;ENDFOLD
;FOLD CIRC CAux389 CDes389 CONT Vel=0.1 m/s CPDATC389 Tool[2] Base[10] ;%{PE}
;FOLD Parameters ;%{h}
;Params IlfProvider=kukaroboter.basistech.inlineforms.movement.old; Kuka.IsGlobalPoint=False; Kuka.PointName=CDes389; Kuka.BlendingEnabled=TRUE; Kuka.MoveDataName=CPDATC389; Kuka.VelocityPath=0.1; Kuka.CurrentCDSetIndex=0; Kuka.MovementParameterFieldEnabled=True; IlfCommand=LIN
;ENDFOLD
$BWDSTART = FALSE
LDAT_ACT=LCPDATC389
FDAT_ACT=FC389
$ORI_TYPE = #VAR
$CIRC_TYPE = #PATH
BAS (#CP_PARAMS,0.1)
SET_CD_PARAMS (0)
CIRC XCAux389, XCDes389 C_DIS

;ENDFOLD
;FOLD LIN P390 CONT Vel=1 m/s CPDATP390 Tool[2] Base[10] ;%{PE}
;FOLD Parameters ;%{h}
;Params IlfProvider=kukaroboter.basistech.inlineforms.movement.old; Kuka.IsGlobalPoint=False; Kuka.PointName=P390; Kuka.BlendingEnabled=TRUE; Kuka.MoveDataName=CPDATP390; Kuka.VelocityPath=1; Kuka.CurrentCDSetIndex=0; Kuka.MovementParameterFieldEnabled=True; IlfCommand=LIN
;ENDFOLD
$BWDSTART = FALSE
LDAT_ACT=LCPDATP390
FDAT_ACT=FP390
BAS (#CP_PARAMS,1)
SET_CD_PARAMS (0)
LIN XP390 C_DIS

;ENDFOLD
;FOLD LIN P391 CONT Vel=1 m/s CPDATP391 Tool[2] Base[10] ;%{PE}
;FOLD Parameters ;%{h}
;Params IlfProvider=kukaroboter.basistech.inlineforms.movement.old; Kuka.IsGlobalPoint=False; Kuka.PointName=P391; Kuka.BlendingEnabled=TRUE; Kuka.MoveDataName=CPDATP391; Kuka.VelocityPath=1; Kuka.CurrentCDSetIndex=0; Kuka.MovementParameterFieldEnabled=True; IlfCommand=LIN
;ENDFOLD
$BWDSTART = FALSE
LDAT_ACT=LCPDATP391
FDAT_ACT=FP391
BAS (#CP_PARAMS,1)
SET_CD_PARAMS (0)
LIN XP391 C_DIS

;ENDFOLD
;FOLD CIRC CAux392 CDes392 CONT Vel=0.1 m/s CPDATC392 Tool[2] Base[10] ;%{PE}
;FOLD Parameters ;%{h}
;Params IlfProvider=kukaroboter.basistech.inlineforms.movement.old; Kuka.IsGlobalPoint=False; Kuka.PointName=CDes392; Kuka.BlendingEnabled=TRUE; Kuka.MoveDataName=CPDATC392; Kuka.VelocityPath=0.1; Kuka.CurrentCDSetIndex=0; Kuka.MovementParameterFieldEnabled=True; IlfCommand=LIN
;ENDFOLD
$BWDSTART = FALSE
LDAT_ACT=LCPDATC392
FDAT_ACT=FC392
$ORI_TYPE = #VAR
$CIRC_TYPE = #PATH
BAS (#CP_PARAMS,0.1)
SET_CD_PARAMS (0)
CIRC XCAux392, XCDes392 C_DIS

;ENDFOLD
;FOLD LIN P393 CONT Vel=1 m/s CPDATP393 Tool[2] Base[10] ;%{PE}
;FOLD Parameters ;%{h}
;Params IlfProvider=kukaroboter.basistech.inlineforms.movement.old; Kuka.IsGlobalPoint=False; Kuka.PointName=P393; Kuka.BlendingEnabled=TRUE; Kuka.MoveDataName=CPDATP393; Kuka.VelocityPath=1; Kuka.CurrentCDSetIndex=0; Kuka.MovementParameterFieldEnabled=True; IlfCommand=LIN
;ENDFOLD
$BWDSTART = FALSE
LDAT_ACT=LCPDATP393
FDAT_ACT=FP393
BAS (#CP_PARAMS,1)
SET_CD_PARAMS (0)
LIN XP393 C_DIS

;ENDFOLD
;FOLD LIN P394 CONT Vel=1 m/s CPDATP394 Tool[2] Base[10] ;%{PE}
;FOLD Parameters ;%{h}
;Params IlfProvider=kukaroboter.basistech.inlineforms.movement.old; Kuka.IsGlobalPoint=False; Kuka.PointName=P394; Kuka.BlendingEnabled=TRUE; Kuka.MoveDataName=CPDATP394; Kuka.VelocityPath=1; Kuka.CurrentCDSetIndex=0; Kuka.MovementParameterFieldEnabled=True; IlfCommand=LIN
;ENDFOLD
$BWDSTART = FALSE
LDAT_ACT=LCPDATP394
FDAT_ACT=FP394
BAS (#CP_PARAMS,1)
SET_CD_PARAMS (0)
LIN XP394 C_DIS

;ENDFOLD
;FOLD CIRC CAux395 CDes395 CONT Vel=0.1 m/s CPDATC395 Tool[2] Base[10] ;%{PE}
;FOLD Parameters ;%{h}
;Params IlfProvider=kukaroboter.basistech.inlineforms.movement.old; Kuka.IsGlobalPoint=False; Kuka.PointName=CDes395; Kuka.BlendingEnabled=TRUE; Kuka.MoveDataName=CPDATC395; Kuka.VelocityPath=0.1; Kuka.CurrentCDSetIndex=0; Kuka.MovementParameterFieldEnabled=True; IlfCommand=LIN
;ENDFOLD
$BWDSTART = FALSE
LDAT_ACT=LCPDATC395
FDAT_ACT=FC395
$ORI_TYPE = #VAR
$CIRC_TYPE = #PATH
BAS (#CP_PARAMS,0.1)
SET_CD_PARAMS (0)
CIRC XCAux395, XCDes395 C_DIS

;ENDFOLD
;FOLD LIN P396 CONT Vel=1 m/s CPDATP396 Tool[2] Base[10] ;%{PE}
;FOLD Parameters ;%{h}
;Params IlfProvider=kukaroboter.basistech.inlineforms.movement.old; Kuka.IsGlobalPoint=False; Kuka.PointName=P396; Kuka.BlendingEnabled=TRUE; Kuka.MoveDataName=CPDATP396; Kuka.VelocityPath=1; Kuka.CurrentCDSetIndex=0; Kuka.MovementParameterFieldEnabled=True; IlfCommand=LIN
;ENDFOLD
$BWDSTART = FALSE
LDAT_ACT=LCPDATP396
FDAT_ACT=FP396
BAS (#CP_PARAMS,1)
SET_CD_PARAMS (0)
LIN XP396 C_DIS

;ENDFOLD
;FOLD LIN P397 CONT Vel=0.5 m/s CPDATP397 Tool[2] Base[10] ;%{PE}
;FOLD Parameters ;%{h}
;Params IlfProvider=kukaroboter.basistech.inlineforms.movement.old; Kuka.IsGlobalPoint=False; Kuka.PointName=P397; Kuka.BlendingEnabled=TRUE; Kuka.MoveDataName=CPDATP397; Kuka.VelocityPath=0.5; Kuka.CurrentCDSetIndex=0; Kuka.MovementParameterFieldEnabled=True; IlfCommand=LIN
;ENDFOLD
$BWDSTART = FALSE
LDAT_ACT=LCPDATP397
FDAT_ACT=FP397
BAS (#CP_PARAMS,0.5)
SET_CD_PARAMS (0)
LIN XP397 C_DIS

;ENDFOLD
;FOLD LIN P398 CONT Vel=0.5 m/s CPDATP398 Tool[2] Base[10] ;%{PE}
;FOLD Parameters ;%{h}
;Params IlfProvider=kukaroboter.basistech.inlineforms.movement.old; Kuka.IsGlobalPoint=False; Kuka.PointName=P398; Kuka.BlendingEnabled=TRUE; Kuka.MoveDataName=CPDATP398; Kuka.VelocityPath=0.5; Kuka.CurrentCDSetIndex=0; Kuka.MovementParameterFieldEnabled=True; IlfCommand=LIN
;ENDFOLD
$BWDSTART = FALSE
LDAT_ACT=LCPDATP398
FDAT_ACT=FP398
BAS (#CP_PARAMS,0.5)
SET_CD_PARAMS (0)
LIN XP398 C_DIS

;ENDFOLD
;FOLD LIN P399 CONT Vel=1.0 m/s CPDATP399 Tool[2] Base[10] ;%{PE}
;FOLD Parameters ;%{h}
;Params IlfProvider=kukaroboter.basistech.inlineforms.movement.old; Kuka.IsGlobalPoint=False; Kuka.PointName=P399; Kuka.BlendingEnabled=TRUE; Kuka.MoveDataName=CPDATP399; Kuka.VelocityPath=1.0; Kuka.CurrentCDSetIndex=0; Kuka.MovementParameterFieldEnabled=True; IlfCommand=LIN
;ENDFOLD
$BWDSTART = FALSE
LDAT_ACT=LCPDATP399
FDAT_ACT=FP399
BAS (#CP_PARAMS,1.0)
SET_CD_PARAMS (0)
LIN XP399 C_DIS

;ENDFOLD
;FOLD LIN P400 CONT Vel=1.0 m/s CPDATP400 Tool[2] Base[10] ;%{PE}
;FOLD Parameters ;%{h}
;Params IlfProvider=kukaroboter.basistech.inlineforms.movement.old; Kuka.IsGlobalPoint=False; Kuka.PointName=P400; Kuka.BlendingEnabled=TRUE; Kuka.MoveDataName=CPDATP400; Kuka.VelocityPath=1.0; Kuka.CurrentCDSetIndex=0; Kuka.MovementParameterFieldEnabled=True; IlfCommand=LIN
;ENDFOLD
$BWDSTART = FALSE
LDAT_ACT=LCPDATP400
FDAT_ACT=FP400
BAS (#CP_PARAMS,1.0)
SET_CD_PARAMS (0)
LIN XP400 C_DIS

;ENDFOLD
END
;End of routine {i}

--- repair_test.dat ---
&ACCESS RVP1
&REL 1217
&PARAM WOPTRAJECTORYID = 2
&PARAM WOPTEMPLATENAME = WopCoreTemplatePath
&PARAM DISKPATH = KRC:\R1\Program\Working Paths
DEFDAT  repair_test
;FOLD EXTERNAL DECLARATIONS;%{PE}%MKUKATPBASIS,%CEXT,%VCOMMON,%P
;FOLD BASISTECH EXT;%{PE}%MKUKATPBASIS,%CEXT,%VEXT,%P
EXT  BAS (BAS_COMMAND  :IN,REAL  :IN )
DECL INT SUCCESS
;ENDFOLD (BASISTECH EXT)
;FOLD USER EXT;%{E}%MKUKATPUSER,%CEXT,%VEXT,%P
;Make your modifications here

;ENDFOLD (USER EXT)
;ENDFOLD (EXTERNAL DECLARATIONS)

INT APP_GENNUMBER = 215375
INT APP_ANSWER
INT APP_OFFSET
DECL STATE_T APP_STATE

DECL PDAT PPDATP0={VEL 100,ACC 100,APO_DIST 5,APO_MODE #CDIS,GEAR_JERK 100.0,EXAX_IGN 0}
DECL FDAT FP0={TOOL_NO 2,BASE_NO 10,IPO_FRAME #BASE,POINT2[] " ",TQ_STATE FALSE}
DECL E6AXIS XP0={A1 -1000.000,A2 -90.000,A3 90.000,A4 0.000,A5 -90.000,A6 0.000,E1 0.000,E2 -41.000,E3 33.000,E4 0.000,E5 0.000,E6 0.000}

; Data for Routine_0
DECL LDAT LCPDATP1={VEL 1,ACC 100,APO_DIST 5,APO_FAC 50.0,ORI_TYP #VAR,CIRC_TYP #BASE,JERK_FAC 50.0}
DECL FDAT FP1={TOOL_NO 2,BASE_NO 10,IPO_FRAME #BASE,POINT2[] " ",TQ_STATE FALSE}
DECL E6POS XP1={X -60.500,Y 111.430,Z -37.190,A 0.000,B -17.860,C -36.410}
DECL LDAT LCPDATC2={VEL 0.1,ACC 100,APO_DIST 5,APO_FAC 50.0,ORI_TYP #VAR,CIRC_TYP #BASE,JERK_FAC 50.0}
DECL FDAT FC2={TOOL_NO 2,BASE_NO 10,IPO_FRAME #BASE,POINT2[] " ",TQ_STATE FALSE}
DECL E6POS XCAux2={X -48.520,Y 117.140,Z -37.190,A 0.000,B -14.240,C -37.780}
DECL E6POS XCDes2={X 48.520,Y 117.140,Z -37.190,A 0.000,B 14.240,C -37.780}
DECL LDAT LCPDATP3={VEL 1,ACC 100,APO_DIST 5,APO_FAC 50.0,ORI_TYP #VAR,CIRC_TYP #BASE,JERK_FAC 50.0}
DECL FDAT FP3={TOOL_NO 2,BASE_NO 10,IPO_FRAME #BASE,POINT2[] " ",TQ_STATE FALSE}
DECL E6POS XP3={X 60.500,Y 111.430,Z -37.190,A 0.000,B 17.860,C -36.410}
DECL LDAT LCPDATP4={VEL 1,ACC 100,APO_DIST 5,APO_FAC 50.0,ORI_TYP #VAR,CIRC_TYP #BASE,JERK_FAC 50.0}
DECL FDAT FP4={TOOL_NO 2,BASE_NO 10,IPO_FRAME #BASE,POINT2[] " ",TQ_STATE FALSE}
DECL E6POS XP4={X 62.870,Y 115.800,Z -40.720,A 0.000,B 14.110,C -27.570}
DECL LDAT LCPDATC5={VEL 0.1,ACC 100,APO_DIST 5,APO_FAC 50.0,ORI_TYP #VAR,CIRC_TYP #BASE,JERK_FAC 50.0}
DECL FDAT FC5={TOOL_NO 2,BASE_NO 10,IPO_FRAME #BASE,POINT2[] " ",TQ_STATE FALSE}
DECL E6POS XCAux5={X 50.420,Y 121.740,Z -40.720,A 0.000,B 11.270,C -28.760}
DECL E6POS XCDes5={X -50.420,Y 121.740,Z -40.720,A 0.000,B -11.270,C -28.760}
DECL LDAT LCPDATP6={VEL 1,ACC 100,APO_DIST 5,APO_FAC 50.0,ORI_TYP #VAR,CIRC_TYP #BASE,JERK_FAC 50.0}
DECL FDAT FP6={TOOL_NO 2,BASE_NO 10,IPO_FRAME #BASE,POINT2[] " ",TQ_STATE FALSE}
DECL E6POS XP6={X -62.870,Y 115.800,Z -40.720,A -0.000,B -14.110,C -27.570}
DECL LDAT LCPDATP7={VEL 1,ACC 100,APO_DIST 5,APO_FAC 50.0,ORI_TYP #VAR,CIRC_TYP #BASE,JERK_FAC 50.0}
DECL FDAT FP7={TOOL_NO 2,BASE_NO 10,IPO_FRAME #BASE,POINT2[] " ",TQ_STATE FALSE}
DECL E6POS XP7={X -65.490,Y 120.610,Z -43.400,A 0.000,B -10.040,C -19.030}
DECL LDAT LCPDATC8={VEL 0.1,ACC 100,APO_DIST 5,APO_FAC 50.0,ORI_TYP #VAR,CIRC_TYP #BASE,JERK_FAC 50.0}
DECL FDAT FC8={TOOL_NO 2,BASE_NO 10,IPO_FRAME #BASE,POINT2[] " ",TQ_STATE FALSE}
DECL E6POS XCAux8={X -52.520,Y 126.790,Z -43.400,A 0.000,B -8.040,C -19.930}
DECL E6POS XCDes8={X 52.520,Y 126.790,Z -43.400,A 0.000,B 8.040,C -19.930}
DECL LDAT LCPDATP9={VEL 1,ACC 100,APO_DIST 5,APO_FAC 50.0,ORI_TYP #VAR,CIRC_TYP #BASE,JERK_FAC 50.0}
DECL FDAT FP9={TOOL_NO 2,BASE_NO 10,IPO_FRAME #BASE,POINT2[] " ",TQ_STATE FALSE}
DECL E6POS XP9={X 65.490,Y 120.610,Z -43.400,A 0.000,B 10.040,C -19.030}
DECL LDAT LCPDATP10={VEL 1,ACC 100,APO_DIST 5,APO_FAC 50.0,ORI_TYP #VAR,CIRC_TYP #BASE,JERK_FAC 50.0}
DECL FDAT FP10={TOOL_NO 2,BASE_NO 10,IPO_FRAME #BASE,POINT2[] " ",TQ_STATE FALSE}
DECL E6POS XP10={X 68.270,Y 125.740,Z -45.160,A -0.000,B 5.760,C -10.710}
DECL LDAT LCPDATC11={VEL 0.1,ACC 100,APO_DIST 5,APO_FAC 50.0,ORI_TYP #VAR,CIRC_TYP #BASE,JERK_FAC 50.0}
DECL FDAT FC11={TOOL_NO 2,BASE_NO 10,IPO_FRAME #BASE,POINT2[] " ",TQ_STATE FALSE}
DECL E6POS XCAux11={X 54.750,Y 132.190,Z -45.160,A -0.000,B 4.620,C -11.250}
DECL E6POS XCDes11={X -54.750,Y 132.190,Z -45.160,A 0.000,B -4.620,C -11.250}
DECL LDAT LCPDATP12={VEL 1,ACC 100,APO_DIST 5,APO_FAC 50.0,ORI_TYP #VAR,CIRC_TYP #BASE,JERK_FAC 50.0}
DECL FDAT FP12={TOOL_NO 2,BASE_NO 10,IPO_FRAME #BASE,POINT2[] " ",TQ_STATE FALSE}
DECL E6POS XP12={X -68.270,Y 125.740,Z -45.160,A 0.000,B -5.760,C -10.710}
DECL LDAT LCPDATP13={VEL 1,ACC 100,APO_DIST 5,APO_FAC 50.0,ORI_TYP #VAR,CIRC_TYP #BASE,JERK_FAC 50.0}
DECL FDAT FP13={TOOL_NO 2,BASE_NO 10,IPO_FRAME #BASE,POINT2[] " ",TQ_STATE FALSE}
DECL E6POS XP13={X -71.150,Y 131.050,Z -45.950,A 0.000,B -1.370,C -2.520}
DECL LDAT LCPDATC14={VEL 0.1,ACC 100,APO_DIST 5,APO_FAC 50.0,ORI_TYP #VAR,CIRC_TYP #BASE,JERK_FAC 50.0}
DECL FDAT FC14={TOOL_NO 2,BASE_NO 10,IPO_FRAME #BASE,POINT2[] " ",TQ_STATE FALSE}
DECL E6POS XCAux14={X -57.070,Y 137.770,Z -45.950,A 0.000,B -1.090,C -2.640}
DECL E6POS XCDes14={X 57.070,Y 137.770,Z -45.950,A -0.000,B 1.090,C -2.640}
DECL LDAT LCPDATP15={VEL 1,ACC 100,APO_DIST 5,APO_FAC 50.0,ORI_TYP #VAR,CIRC_TYP #BASE,JERK_FAC 50.0}
DECL FDAT FP15={TOOL_NO 2,BASE_NO 10,IPO_FRAME #BASE,POINT2[] " ",TQ_STATE FALSE}
DECL E6POS XP15={X 71.150,Y 131.050,Z -45.950,A 0.000,B 1.370,C -2.520}
DECL LDAT LCPDATP16={VEL 1,ACC 100,APO_DIST 5,APO_FAC 50.0,ORI_TYP #VAR,CIRC_TYP #BASE,JERK_FAC 50.0}
DECL FDAT FP16={TOOL_NO 2,BASE_NO 10,IPO_FRAME #BASE,POINT2[] " ",TQ_STATE FALSE}
DECL E6POS XP16={X 71.390,Y 131.490,Z -46.000,A 0.000,B 0.000,C -0.000}
DECL LDAT LCPDATC17={VEL 0.1,ACC 100,APO_DIST 5,APO_FAC 50.0,ORI_TYP #VAR,CIRC_TYP #BASE,JERK_FAC 50.0}
DECL FDAT FC17={TOOL_NO 2,BASE_NO 10,IPO_FRAME #BASE,POINT2[] " ",TQ_STATE FALSE}
DECL E6POS XCAux17={X 57.260,Y 138.230,Z -46.000,A 0.000,B 0.000,C -0.000}
DECL E6POS XCDes17={X -57.260,Y 138.230,Z -46.000,A 0.000,B 0.000,C -0.000}
DECL LDAT LCPDATP18={VEL 1,ACC 100,APO_DIST 5,APO_FAC 50.0,ORI_TYP #VAR,CIRC_TYP #BASE,JERK_FAC 50.0}
DECL FDAT FP18={TOOL_NO 2,BASE_NO 10,IPO_FRAME #BASE,POINT2[] " ",TQ_STATE FALSE}
DECL E6POS XP18={X -71.390,Y 131.490,Z -46.000,A 0.000,B 0.000,C -0.000}
DECL LDAT LCPDATP19={VEL 1,ACC 100,APO_DIST 5,APO_FAC 50.0,ORI_TYP #VAR,CIRC_TYP #BASE,JERK_FAC 50.0}
DECL FDAT FP19={TOOL_NO 2,BASE_NO 10,IPO_FRAME #BASE,POINT2[] " ",TQ_STATE FALSE}
DECL E6POS XP19={X -70.440,Y 129.730,Z -46.000,A 0.000,B 0.000,C -0.000}
DECL LDAT LCPDATC20={VEL 0.1,ACC 100,APO_DIST 5,APO_FAC 50.0,ORI_TYP #VAR,CIRC_TYP #BASE,JERK_FAC 50.0}
DECL FDAT FC20={TOOL_NO 2,BASE_NO 10,IPO_FRAME #BASE,POINT2[] " ",TQ_STATE FALSE}
DECL E6POS XCAux20={X -56.490,Y 136.380,Z -46.000,A 0.000,B 0.000,C -0.000}
DECL E6POS XCDes20={X 56.490,Y 136.380,Z -46.000,A 0.000,B 0.000,C -0.000}
DECL LDAT LCPDATP21={VEL 1,ACC 100,APO_DIST 5,APO_FAC 50.0,ORI_TYP #VAR,CIRC_TYP #BASE,JERK_FAC 50.0}
DECL FDAT FP21={TOOL_NO 2,BASE_NO 10,IPO_FRAME #BASE,POINT2[] " ",TQ_STATE FALSE}
DECL E6POS XP21={X 70.440,Y 129.730,Z -46.000,A 0.000,B 0.000,C -0.000}
DECL LDAT LCPDATP22={VEL 1,ACC 100,APO_DIST 5,APO_FAC 50.0,ORI_TYP #VAR,CIRC_TYP #BASE,JERK_FAC 50.0}
DECL FDAT FP22={TOOL_NO 2,BASE_NO 10,IPO_FRAME #BASE,POINT2[] " ",TQ_STATE FALSE}
DECL E6POS XP22={X 69.480,Y 127.970,Z -46.000,A 0.000,B 0.000,C -0.000}
DECL LDAT LCPDATC23={VEL 0.1,ACC 100,APO_DIST 5,APO_FAC 50.0,ORI_TYP #VAR,CIRC_TYP #BASE,JERK_FAC 50.0}
DECL FDAT FC23={TOOL_NO 2,BASE_NO 10,IPO_FRAME #BASE,POINT2[] " ",TQ_STATE FALSE}
DECL E6POS XCAux23={X 55.720,Y 134.530,Z -46.000,A 0.000,B 0.000,C -0.000}
DECL E6POS XCDes23={X -55.720,Y 134.530,Z -46.000,A 0.000,B 0.000,C -0.000}
DECL LDAT LCPDATP24={VEL 1,ACC 100,APO_DIST 5,APO_FAC 50.0,ORI_TYP #VAR,CIRC_TYP #BASE,JERK_FAC 50.0}
DECL FDAT FP24={TOOL_NO 2,BASE_NO 10,IPO_FRAME #BASE,POINT2[] " ",TQ_STATE FALSE}
DECL E6POS XP24={X -69.480,Y 127.970,Z -46.000,A 0.000,B 0.000,C -0.000}
DECL LDAT LCPDATP25={VEL 1,ACC 100,APO_DIST 5,APO_FAC 50.0,ORI_TYP #VAR,CIRC_TYP #BASE,JERK_FAC 50.0}
DECL FDAT FP25={TOOL_NO 2,BASE_NO 10,IPO_FRAME #BASE,POINT2[] " ",TQ_STATE FALSE}
DECL E6POS XP25={X -68.530,Y 126.210,Z -46.000,A 0.000,B 0.000,C -0.000}
DECL LDAT LCPDATC26={VEL 0.1,ACC 100,APO_DIST 5,APO_FAC 50.0,ORI_TYP #VAR,CIRC_TYP #BASE,JERK_FAC 50.0}
DECL FDAT FC26={TOOL_NO 2,BASE_NO 10,IPO_FRAME #BASE,POINT2[] " ",TQ_STATE FALSE}
DECL E6POS XCAux26={X -54.960,Y 132.680,Z -46.000,A 0.000,B 0.000,C -0.000}
DECL E6POS XCDes26={X 54.960,Y 132.680,Z -46.000,A 0.000,B 0.000,C -0.000}
DECL LDAT LCPDATP27={VEL 1,ACC 100,APO_DIST 5,APO_FAC 50.0,ORI_TYP #VAR,CIRC_TYP #BASE,JERK_FAC 50.0}
DECL FDAT FP27={TOOL_NO 2,BASE_NO 10,IPO_FRAME #BASE,POINT2[] " ",TQ_STATE FALSE}
DECL E6POS XP27={X 68.530,Y 126.210,Z -46.000,A 0.000,B 0.000,C -0.000}
DECL LDAT LCPDATP28={VEL 1,ACC 100,APO_DIST 5,APO_FAC 50.0,ORI_TYP #VAR,CIRC_TYP #BASE,JERK_FAC 50.0}
DECL FDAT FP28={TOOL_NO 2,BASE_NO 10,IPO_FRAME #BASE,POINT2[] " ",TQ_STATE FALSE}
DECL E6POS XP28={X 67.570,Y 124.450,Z -46.000,A 0.000,B 0.000,C -0.000}
DECL LDAT LCPDATC29={VEL 0.1,ACC 100,APO_DIST 5,APO_FAC 50.0,ORI_TYP #VAR,CIRC_TYP #BASE,JERK_FAC 50.0}
DECL FDAT FC29={TOOL_NO 2,BASE_NO 10,IPO_FRAME #BASE,POINT2[] " ",TQ_STATE FALSE}
DECL E6POS XCAux29={X 54.190,Y 130.840,Z -46.000,A 0.000,B 0.000,C -0.000}
DECL E6POS XCDes29={X -54.190,Y 130.840,Z -46.000,A 0.000,B 0.000,C -0.000}
DECL LDAT LCPDATP30={VEL 1,ACC 100,APO_DIST 5,APO_FAC 50.0,ORI_TYP #VAR,CIRC_TYP #BASE,JERK_FAC 50.0}
DECL FDAT FP30={TOOL_NO 2,BASE_NO 10,IPO_FRAME #BASE,POINT2[] " ",TQ_STATE FALSE}
DECL E6POS XP30={X -67.570,Y 124.450,Z -46.000,A 0.000,B 0.000,C -0.000}
DECL LDAT LCPDATP31={VEL 1,ACC 100,APO_DIST 5,APO_FAC 50.0,ORI_TYP #VAR,CIRC_TYP #BASE,JERK_FAC 50.0}
DECL FDAT FP31={TOOL_NO 2,BASE_NO 10,IPO_FRAME #BASE,POINT2[] " ",TQ_STATE FALSE}
DECL E6POS XP31={X -66.620,Y 122.700,Z -46.000,A 0.000,B 0.000,C -0.000}
DECL LDAT LCPDATC32={VEL 0.1,ACC 100,APO_DIST 5,APO_FAC 50.0,ORI_TYP #VAR,CIRC_TYP #BASE,JERK_FAC 50.0}
DECL FDAT FC32={TOOL_NO 2,BASE_NO 10,IPO_FRAME #BASE,POINT2[] " ",TQ_STATE FALSE}
DECL E6POS XCAux32={X -53.430,Y 128.990,Z -46.000,A 0.000,B 0.000,C -0.000}
DECL E6POS XCDes32={X 53.430,Y 128.990,Z -46.000,A 0.000,B 0.000,C -0.000}
DECL LDAT LCPDATP33={VEL 1,ACC 100,APO_DIST 5,APO_FAC 50.0,ORI_TYP #VAR,CIRC_TYP #BASE,JERK_FAC 50.0}
DECL FDAT FP33={TOOL_NO 2,BASE_NO 10,IPO_FRAME #BASE,POINT2[] " ",TQ_STATE FALSE}
DECL E6POS XP33={X 66.620,Y 122.700,Z -46.000,A 0.000,B 0.000,C -0.000}
DECL LDAT LCPDATP34={VEL 1,ACC 100,APO_DIST 5,APO_FAC 50.0,ORI_TYP #VAR,CIRC_TYP #BASE,JERK_FAC 50.0}
DECL FDAT FP34={TOOL_NO 2,BASE_NO 10,IPO_FRAME #BASE,POINT2[] " ",TQ_STATE FALSE}
DECL E6POS XP34={X 68.340,Y 125.870,Z -45.760,A 0.000,B -3.070,C 5.660}
DECL LDAT LCPDATC35={VEL 0.1,ACC 100,APO_DIST 5,APO_FAC 50.0,ORI_TYP #VAR,CIRC_TYP #BASE,JERK_FAC 50.0}
DECL FDAT FC35={TOOL_NO 2,BASE_NO 10,IPO_FRAME #BASE,POINT2[] " ",TQ_STATE FALSE}
DECL E6POS XCAux35={X 54.810,Y 132.320,Z -45.760,A -0.000,B -2.460,C 5.950}
DECL E6POS XCDes35={X -54.810,Y 132.320,Z -45.760,A 0.000,B 2.460,C 5.950}
DECL LDAT LCPDATP36={VEL 1,ACC 100,APO_DIST 5,APO_FAC 50.0,ORI_TYP #VAR,CIRC_TYP #BASE,JERK_FAC 50.0}
DECL FDAT FP36={TOOL_NO 2,BASE_NO 10,IPO_FRAME #BASE,POINT2[] " ",TQ_STATE FALSE}
DECL E6POS XP36={X -68.340,Y 125.870,Z -45.760,A 0.000,B 3.070,C 5.660}
DECL LDAT LCPDATP37={VEL 1,ACC 100,APO_DIST 5,APO_FAC 50.0,ORI_TYP #VAR,CIRC_TYP #BASE,JERK_FAC 50.0}
DECL FDAT FP37={TOOL_NO 2,BASE_NO 10,IPO_FRAME #BASE,POINT2[] " ",TQ_STATE FALSE}
DECL E6POS XP37={X -71.190,Y 131.120,Z -44.590,A 0.000,B 7.430,C 13.890}
DECL LDAT LCPDATC38={VEL 0.1,ACC 100,APO_DIST 5,APO_FAC 50.0,ORI_TYP #VAR,CIRC_TYP #BASE,JERK_FAC 50.0}
DECL FDAT FC38={TOOL_NO 2,BASE_NO 10,IPO_FRAME #BASE,POINT2[] " ",TQ_STATE FALSE}
DECL E6POS XCAux38={X -57.100,Y 137.850,Z -44.590,A -0.000,B 5.950,C 14.580}
DECL E6POS XCDes38={X 57.100,Y 137.850,Z -44.590,A 0.000,B -5.950,C 14.580}
DECL LDAT LCPDATP39={VEL 1,ACC 100,APO_DIST 5,APO_FAC 50.0,ORI_TYP #VAR,CIRC_TYP #BASE,JERK_FAC 50.0}
DECL FDAT FP39={TOOL_NO 2,BASE_NO 10,IPO_FRAME #BASE,POINT2[] " ",TQ_STATE FALSE}
DECL E6POS XP39={X 71.190,Y 131.120,Z -44.590,A 0.000,B -7.430,C 13.890}
DECL LDAT LCPDATP40={VEL 1,ACC 100,APO_DIST 5,APO_FAC 50.0,ORI_TYP #VAR,CIRC_TYP #BASE,JERK_FAC 50.0}
DECL FDAT FP40={TOOL_NO 2,BASE_NO 10,IPO_FRAME #BASE,POINT2[] " ",TQ_STATE FALSE}
DECL E6POS XP40={X 73.920,Y 136.140,Z -42.470,A -0.000,B -11.640,C 22.290}
DECL LDAT LCPDATC41={VEL 0.1,ACC 100,APO_DIST 5,APO_FAC 50.0,ORI_TYP #VAR,CIRC_TYP #BASE,JERK_FAC 50.0}
DECL FDAT FC41={TOOL_NO 2,BASE_NO 10,IPO_FRAME #BASE,POINT2[] " ",TQ_STATE FALSE}
DECL E6POS XCAux41={X 59.280,Y 143.130,Z -42.470,A 0.000,B -9.310,C 23.310}
DECL E6POS XCDes41={X -59.280,Y 143.130,Z -42.470,A 0.000,B 9.310,C 23.310}
DECL LDAT LCPDATP42={VEL 1,ACC 100,APO_DIST 5,APO_FAC 50.0,ORI_TYP #VAR,CIRC_TYP #BASE,JERK_FAC 50.0}
DECL FDAT FP42={TOOL_NO 2,BASE_NO 10,IPO_FRAME #BASE,POINT2[] " ",TQ_STATE FALSE}
DECL E6POS XP42={X -73.920,Y 136.140,Z -42.470,A 0.000,B 11.640,C 22.290}
DECL LDAT LCPDATP43={VEL 1,ACC 100,APO_DIST 5,APO_FAC 50.0,ORI_TYP #VAR,CIRC_TYP #BASE,JERK_FAC 50.0}
DECL FDAT FP43={TOOL_NO 2,BASE_NO 10,IPO_FRAME #BASE,POINT2[] " ",TQ_STATE FALSE}
DECL E6POS XP43={X -76.450,Y 140.800,Z -39.450,A -0.000,B 15.590,C 30.930}
DECL LDAT LCPDATC44={VEL 0.1,ACC 100,APO_DIST 5,APO_FAC 50.0,ORI_TYP #VAR,CIRC_TYP #BASE,JERK_FAC 50.0}
DECL FDAT FC44={TOOL_NO 2,BASE_NO 10,IPO_FRAME #BASE,POINT2[] " ",TQ_STATE FALSE}
DECL E6POS XCAux44={X -61.310,Y 148.020,Z -39.450,A 0.000,B 12.450,C 32.210}
DECL E6POS XCDes44={X 61.310,Y 148.020,Z -39.450,A -0.000,B -12.450,C 32.210}
DECL LDAT LCPDATP45={VEL 1,ACC 100,APO_DIST 5,APO_FAC 50.0,ORI_TYP #VAR,CIRC_TYP #BASE,JERK_FAC 50.0}
DECL FDAT FP45={TOOL_NO 2,BASE_NO 10,IPO_FRAME #BASE,POINT2[] " ",TQ_STATE FALSE}
DECL E6POS XP45={X 76.450,Y 140.800,Z -39.450,A 0.000,B -15.590,C 30.930}
DECL LDAT LCPDATP46={VEL 1,ACC 100,APO_DIST 5,APO_FAC 50.0,ORI_TYP #VAR,CIRC_TYP #BASE,JERK_FAC 50.0}
DECL FDAT FP46={TOOL_NO 2,BASE_NO 10,IPO_FRAME #BASE,POINT2[] " ",TQ_STATE FALSE}
DECL E6POS XP46={X 78.710,Y 144.970,Z -35.620,A -0.000,B -19.200,C 39.900}
DECL LDAT LCPDATC47={VEL 0.1,ACC 100,APO_DIST 5,APO_FAC 50.0,ORI_TYP #VAR,CIRC_TYP #BASE,JERK_FAC 50.0}
DECL FDAT FC47={TOOL_NO 2,BASE_NO 10,IPO_FRAME #BASE,POINT2[] " ",TQ_STATE FALSE}
DECL E6POS XCAux47={X 63.130,Y 152.400,Z -35.620,A -0.000,B -15.290,C 41.320}
DECL E6POS XCDes47={X -63.130,Y 152.400,Z -35.620,A -0.000,B 15.290,C 41.320}
DECL LDAT LCPDATP48={VEL 1,ACC 100,APO_DIST 5,APO_FAC 50.0,ORI_TYP #VAR,CIRC_TYP #BASE,JERK_FAC 50.0}
DECL FDAT FP48={TOOL_NO 2,BASE_NO 10,IPO_FRAME #BASE,POINT2[] " ",TQ_STATE FALSE}
DECL E6POS XP48={X -78.710,Y 144.970,Z -35.620,A 0.000,B 19.200,C 39.900}
DECL LDAT LCPDATP49={VEL 1,ACC 100,APO_DIST 5,APO_FAC 50.0,ORI_TYP #VAR,CIRC_TYP #BASE,JERK_FAC 50.0}
DECL FDAT FP49={TOOL_NO 2,BASE_NO 10,IPO_FRAME #BASE,POINT2[] " ",TQ_STATE FALSE}
DECL E6POS XP49={X -78.000,Y 143.650,Z -37.500,A -0.000,B 17.860,C 36.410}
DECL LDAT LCPDATC50={VEL 0.1,ACC 100,APO_DIST 5,APO_FAC 50.0,ORI_TYP #VAR,CIRC_TYP #BASE,JERK_FAC 50.0}
DECL FDAT FC50={TOOL_NO 2,BASE_NO 10,IPO_FRAME #BASE,POINT2[] " ",TQ_STATE FALSE}
DECL E6POS XCAux50={X -62.550,Y 151.020,Z -37.500,A -0.000,B 14.240,C 37.780}
DECL E6POS XCDes50={X 62.550,Y 151.020,Z -37.500,A 0.000,B -14.240,C 37.780}
DECL LDAT LCPDATP51={VEL 1,ACC 100,APO_DIST 5,APO_FAC 50.0,ORI_TYP #VAR,CIRC_TYP #BASE,JERK_FAC 50.0}
DECL FDAT FP51={TOOL_NO 2,BASE_NO 10,IPO_FRAME #BASE,POINT2[] " ",TQ_STATE FALSE}
DECL E6POS XP51={X 78.000,Y 143.650,Z -37.500,A -0.000,B -17.860,C 36.410}
DECL LDAT LCPDATP52={VEL 1,ACC 100,APO_DIST 5,APO_FAC 50.0,ORI_TYP #VAR,CIRC_TYP #BASE,JERK_FAC 50.0}
DECL FDAT FP52={TOOL_NO 2,BASE_NO 10,IPO_FRAME #BASE,POINT2[] " ",TQ_STATE FALSE}
DECL E6POS XP52={X 75.520,Y 139.080,Z -41.170,A -0.000,B -13.970,C 27.280}
DECL LDAT LCPDATC53={VEL 0.1,ACC 100,APO_DIST 5,APO_FAC 50.0,ORI_TYP #VAR,CIRC_TYP #BASE,JERK_FAC 50.0}
DECL FDAT FC53={TOOL_NO 2,BASE_NO 10,IPO_FRAME #BASE,POINT2[] " ",TQ_STATE FALSE}
DECL E6POS XCAux53={X 60.560,Y 146.210,Z -41.170,A 0.000,B -11.170,C 28.460}
DECL E6POS XCDes53={X -60.560,Y 146.210,Z -41.170,A -0.000,B 11.170,C 28.460}
DECL LDAT LCPDATP54={VEL 1,ACC 100,APO_DIST 5,APO_FAC 50.0,ORI_TYP #VAR,CIRC_TYP #BASE,JERK_FAC 50.0}
DECL FDAT FP54={TOOL_NO 2,BASE_NO 10,IPO_FRAME #BASE,POINT2[] " ",TQ_STATE FALSE}
DECL E6POS XP54={X -75.520,Y 139.080,Z -41.170,A 0.000,B 13.970,C 27.280}
DECL LDAT LCPDATP55={VEL 1,ACC 100,APO_DIST 5,APO_FAC 50.0,ORI_TYP #VAR,CIRC_TYP #BASE,JERK_FAC 50.0}
DECL FDAT FP55={TOOL_NO 2,BASE_NO 10,IPO_FRAME #BASE,POINT2[] " ",TQ_STATE FALSE}
DECL E6POS XP55={X -72.780,Y 134.040,Z -43.920,A 0.000,B 9.760,C 18.470}
DECL LDAT LCPDATC56={VEL 0.1,ACC 100,APO_DIST 5,APO_FAC 50.0,ORI_TYP #VAR,CIRC_TYP #BASE,JERK_FAC 50.0}
DECL FDAT FC56={TOOL_NO 2,BASE_NO 10,IPO_FRAME #BASE,POINT2[] " ",TQ_STATE FALSE}
DECL E6POS XCAux56={X -58.370,Y 140.910,Z -43.920,A 0.000,B 7.810,C 19.350}
DECL E6POS XCDes56={X 58.370,Y 140.910,Z -43.920,A -0.000,B -7.810,C 19.350}
DECL LDAT LCPDATP57={VEL 1,ACC 100,APO_DIST 5,APO_FAC 50.0,ORI_TYP #VAR,CIRC_TYP #BASE,JERK_FAC 50.0}
DECL FDAT FP57={TOOL_NO 2,BASE_NO 10,IPO_FRAME #BASE,POINT2[] " ",TQ_STATE FALSE}
DECL E6POS XP57={X 72.780,Y 134.040,Z -43.920,A 0.000,B -9.760,C 18.470}
DECL LDAT LCPDATP58={VEL 1,ACC 100,APO_DIST 5,APO_FAC 50.0,ORI_TYP #VAR,CIRC_TYP #BASE,JERK_FAC 50.0}
DECL FDAT FP58={TOOL_NO 2,BASE_NO 10,IPO_FRAME #BASE,POINT2[] " ",TQ_STATE FALSE}
DECL E6POS XP58={X 69.860,Y 128.660,Z -45.670,A -0.000,B -5.320,C 9.880}
DECL LDAT LCPDATC59={VEL 0.1,ACC 100,APO_DIST 5,APO_FAC 50.0,ORI_TYP #VAR,CIRC_TYP #BASE,JERK_FAC 50.0}
DECL FDAT FC59={TOOL_NO 2,BASE_NO 10,IPO_FRAME #BASE,POINT2[] " ",TQ_STATE FALSE}
DECL E6POS XCAux59={X 56.030,Y 135.260,Z -45.670,A -0.000,B -4.270,C 10.380}
DECL E6POS XCDes59={X -56.030,Y 135.260,Z -45.670,A -0.000,B 4.270,C 10.380}
DECL LDAT LCPDATP60={VEL 1,ACC 100,APO_DIST 5,APO_FAC 50.0,ORI_TYP #VAR,CIRC_TYP #BASE,JERK_FAC 50.0}
DECL FDAT FP60={TOOL_NO 2,BASE_NO 10,IPO_FRAME #BASE,POINT2[] " ",TQ_STATE FALSE}
DECL E6POS XP60={X -69.860,Y 128.660,Z -45.670,A 0.000,B 5.320,C 9.880}
DECL LDAT LCPDATP61={VEL 1,ACC 100,APO_DIST 5,APO_FAC 50.0,ORI_TYP #VAR,CIRC_TYP #BASE,JERK_FAC 50.0}
DECL FDAT FP61={TOOL_NO 2,BASE_NO 10,IPO_FRAME #BASE,POINT2[] " ",TQ_STATE FALSE}
DECL E6POS XP61={X -66.840,Y 123.100,Z -46.380,A 0.000,B 0.770,C 1.420}
DECL LDAT LCPDATC62={VEL 0.1,ACC 100,APO_DIST 5,APO_FAC 50.0,ORI_TYP #VAR,CIRC_TYP #BASE,JERK_FAC 50.0}
DECL FDAT FC62={TOOL_NO 2,BASE_NO 10,IPO_FRAME #BASE,POINT2[] " ",TQ_STATE FALSE}
DECL E6POS XCAux62={X -53.600,Y 129.410,Z -46.380,A 0.000,B 0.620,C 1.500}
DECL E6POS XCDes62={X 53.600,Y 129.410,Z -46.380,A 0.000,B -0.620,C 1.500}
DECL LDAT LCPDATP63={VEL 1,ACC 100,APO_DIST 5,APO_FAC 50.0,ORI_TYP #VAR,CIRC_TYP #BASE,JERK_FAC 50.0}
DECL FDAT FP63={TOOL_NO 2,BASE_NO 10,IPO_FRAME #BASE,POINT2[] " ",TQ_STATE FALSE}
DECL E6POS XP63={X 66.840,Y 123.100,Z -46.380,A 0.000,B -0.770,C 1.420}
DECL LDAT LCPDATP64={VEL 1,ACC 100,APO_DIST 5,APO_FAC 50.0,ORI_TYP #VAR,CIRC_TYP #BASE,JERK_FAC 50.0}
DECL FDAT FP64={TOOL_NO 2,BASE_NO 10,IPO_FRAME #BASE,POINT2[] " ",TQ_STATE FALSE}
DECL E6POS XP64={X 67.120,Y 123.620,Z -46.400,A 0.000,B 0.000,C -0.000}
DECL LDAT LCPDATC65={VEL 0.1,ACC 100,APO_DIST 5,APO_FAC 50.0,ORI_TYP #VAR,CIRC_TYP #BASE,JERK_FAC 50.0}
DECL FDAT FC65={TOOL_NO 2,BASE_NO 10,IPO_FRAME #BASE,POINT2[] " ",TQ_STATE FALSE}
DECL E6POS XCAux65={X 53.830,Y 129.960,Z -46.400,A 0.000,B 0.000,C -0.000}
DECL E6POS XCDes65={X -53.830,Y 129.960,Z -46.400,A 0.000,B 0.000,C -0.000}
DECL LDAT LCPDATP66={VEL 1,ACC 100,APO_DIST 5,APO_FAC 50.0,ORI_TYP #VAR,CIRC_TYP #BASE,JERK_FAC 50.0}
DECL FDAT FP66={TOOL_NO 2,BASE_NO 10,IPO_FRAME #BASE,POINT2[] " ",TQ_STATE FALSE}
DECL E6POS XP66={X -67.120,Y 123.620,Z -46.400,A 0.000,B 0.000,C -0.000}
DECL LDAT LCPDATP67={VEL 1,ACC 100,APO_DIST 5,APO_FAC 50.0,ORI_TYP #VAR,CIRC_TYP #BASE,JERK_FAC 50.0}
DECL FDAT FP67={TOOL_NO 2,BASE_NO 10,IPO_FRAME #BASE,POINT2[] " ",TQ_STATE FALSE}
DECL E6POS XP67={X -68.070,Y 125.370,Z -46.400,A 0.000,B 0.000,C -0.000}
DECL LDAT LCPDATC68={VEL 0.1,ACC 100,APO_DIST 5,APO_FAC 50.0,ORI_TYP #VAR,CIRC_TYP #BASE,JERK_FAC 50.0}
DECL FDAT FC68={TOOL_NO 2,BASE_NO 10,IPO_FRAME #BASE,POINT2[] " ",TQ_STATE FALSE}
DECL E6POS XCAux68={X -54.590,Y 131.800,Z -46.400,A 0.000,B 0.000,C -0.000}
DECL E6POS XCDes68={X 54.590,Y 131.800,Z -46.400,A 0.000,B 0.000,C -0.000}
DECL LDAT LCPDATP69={VEL 1,ACC 100,APO_DIST 5,APO_FAC 50.0,ORI_TYP #VAR,CIRC_TYP #BASE,JERK_FAC 50.0}
DECL FDAT FP69={TOOL_NO 2,BASE_NO 10,IPO_FRAME #BASE,POINT2[] " ",TQ_STATE FALSE}
DECL E6POS XP69={X 68.070,Y 125.370,Z -46.400,A 0.000,B 0.000,C -0.000}
DECL LDAT LCPDATP70={VEL 1,ACC 100,APO_DIST 5,APO_FAC 50.0,ORI_TYP #VAR,CIRC_TYP #BASE,JERK_FAC 50.0}
DECL FDAT FP70={TOOL_NO 2,BASE_NO 10,IPO_FRAME #BASE,POINT2[] " ",TQ_STATE FALSE}
DECL E6POS XP70={X 69.030,Y 127.130,Z -46.400,A 0.000,B 0.000,C -0.000}
DECL LDAT LCPDATC71={VEL 0.1,ACC 100,APO_DIST 5,APO_FAC 50.0,ORI_TYP #VAR,CIRC_TYP #BASE,JERK_FAC 50.0}
DECL FDAT FC71={TOOL_NO 2,BASE_NO 10,IPO_FRAME #BASE,POINT2[] " ",TQ_STATE FALSE}
DECL E6POS XCAux71={X 55.360,Y 133.650,Z -46.400,A 0.000,B 0.000,C -0.000}
DECL E6POS XCDes71={X -55.360,Y 133.650,Z -46.400,A 0.000,B 0.000,C -0.000}
DECL LDAT LCPDATP72={VEL 1,ACC 100,APO_DIST 5,APO_FAC 50.0,ORI_TYP #VAR,CIRC_TYP #BASE,JERK_FAC 50.0}
DECL FDAT FP72={TOOL_NO 2,BASE_NO 10,IPO_FRAME #BASE,POINT2[] " ",TQ_STATE FALSE}
DECL E6POS XP72={X -69.030,Y 127.130,Z -46.400,A 0.000,B 0.000,C -0.000}
DECL LDAT LCPDATP73={VEL 1,ACC 100,APO_DIST 5,APO_FAC 50.0,ORI_TYP #VAR,CIRC_TYP #BASE,JERK_FAC 50.0}
DECL FDAT FP73={TOOL_NO 2,BASE_NO 10,IPO_FRAME #BASE,POINT2[] " ",TQ_STATE FALSE}
DECL E6POS XP73={X -69.980,Y 128.890,Z -46.400,A 0.000,B 0.000,C -0.000}
DECL LDAT LCPDATC74={VEL 0.1,ACC 100,APO_DIST 5,APO_FAC 50.0,ORI_TYP #VAR,CIRC_TYP #BASE,JERK_FAC 50.0}
DECL FDAT FC74={TOOL_NO 2,BASE_NO 10,IPO_FRAME #BASE,POINT2[] " ",TQ_STATE FALSE}
DECL E6POS XCAux74={X -56.130,Y 135.500,Z -46.400,A 0.000,B 0.000,C -0.000}
DECL E6POS XCDes74={X 56.130,Y 135.500,Z -46.400,A 0.000,B 0.000,C -0.000}
DECL LDAT LCPDATP75={VEL 1,ACC 100,APO_DIST 5,APO_FAC 50.0,ORI_TYP #VAR,CIRC_TYP #BASE,JERK_FAC 50.0}
DECL FDAT FP75={TOOL_NO 2,BASE_NO 10,IPO_FRAME #BASE,POINT2[] " ",TQ_STATE FALSE}
DECL E6POS XP75={X 69.980,Y 128.890,Z -46.400,A 0.000,B 0.000,C -0.000}
DECL LDAT LCPDATP76={VEL 1,ACC 100,APO_DIST 5,APO_FAC 50.0,ORI_TYP #VAR,CIRC_TYP #BASE,JERK_FAC 50.0}
DECL FDAT FP76={TOOL_NO 2,BASE_NO 10,IPO_FRAME #BASE,POINT2[] " ",TQ_STATE FALSE}
DECL E6POS XP76={X 70.940,Y 130.650,Z -46.400,A 0.000,B 0.000,C -0.000}
DECL LDAT LCPDATC77={VEL 0.1,ACC 100,APO_DIST 5,APO_FAC 50.0,ORI_TYP #VAR,CIRC_TYP #BASE,JERK_FAC 50.0}
DECL FDAT FC77={TOOL_NO 2,BASE_NO 10,IPO_FRAME #BASE,POINT2[] " ",TQ_STATE FALSE}
DECL E6POS XCAux77={X 56.890,Y 137.350,Z -46.400,A 0.000,B 0.000,C -0.000}
DECL E6POS XCDes77={X -56.890,Y 137.350,Z -46.400,A 0.000,B 0.000,C -0.000}
DECL LDAT LCPDATP78={VEL 1,ACC 100,APO_DIST 5,APO_FAC 50.0,ORI_TYP #VAR,CIRC_TYP #BASE,JERK_FAC 50.0}
DECL FDAT FP78={TOOL_NO 2,BASE_NO 10,IPO_FRAME #BASE,POINT2[] " ",TQ_STATE FALSE}
DECL E6POS XP78={X -70.940,Y 130.650,Z -46.400,A 0.000,B 0.000,C -0.000}
DECL LDAT LCPDATP79={VEL 1,ACC 100,APO_DIST 5,APO_FAC 50.0,ORI_TYP #VAR,CIRC_TYP #BASE,JERK_FAC 50.0}
DECL FDAT FP79={TOOL_NO 2,BASE_NO 10,IPO_FRAME #BASE,POINT2[] " ",TQ_STATE FALSE}
DECL E6POS XP79={X -71.890,Y 132.410,Z -46.400,A 0.000,B 0.000,C -0.000}
DECL LDAT LCPDATC80={VEL 0.1,ACC 100,APO_DIST 5,APO_FAC 50.0,ORI_TYP #VAR,CIRC_TYP #BASE,JERK_FAC 50.0}
DECL FDAT FC80={TOOL_NO 2,BASE_NO 10,IPO_FRAME #BASE,POINT2[] " ",TQ_STATE FALSE}
DECL E6POS XCAux80={X -57.660,Y 139.190,Z -46.400,A 0.000,B 0.000,C -0.000}
DECL E6POS XCDes80={X 57.660,Y 139.190,Z -46.400,A 0.000,B 0.000,C -0.000}
DECL LDAT LCPDATP81={VEL 1,ACC 100,APO_DIST 5,APO_FAC 50.0,ORI_TYP #VAR,CIRC_TYP #BASE,JERK_FAC 50.0}
DECL FDAT FP81={TOOL_NO 2,BASE_NO 10,IPO_FRAME #BASE,POINT2[] " ",TQ_STATE FALSE}
DECL E6POS XP81={X 71.890,Y 132.410,Z -46.400,A 0.000,B 0.000,C -0.000}
DECL LDAT LCPDATP82={VEL 1,ACC 100,APO_DIST 5,APO_FAC 50.0,ORI_TYP #VAR,CIRC_TYP #BASE,JERK_FAC 50.0}
DECL FDAT FP82={TOOL_NO 2,BASE_NO 10,IPO_FRAME #BASE,POINT2[] " ",TQ_STATE FALSE}
DECL E6POS XP82={X 69.520,Y 128.040,Z -46.030,A -0.000,B 3.810,C -7.040}
DECL LDAT LCPDATC83={VEL 0.1,ACC 100,APO_DIST 5,APO_FAC 50.0,ORI_TYP #VAR,CIRC_TYP #BASE,JERK_FAC 50.0}
DECL FDAT FC83={TOOL_NO 2,BASE_NO 10,IPO_FRAME #BASE,POINT2[] " ",TQ_STATE FALSE}
DECL E6POS XCAux83={X 55.760,Y 134.610,Z -46.030,A 0.000,B 3.050,C -7.400}
DECL E6POS XCDes83={X -55.760,Y 134.610,Z -46.030,A -0.000,B -3.050,C -7.400}
DECL LDAT LCPDATP84={VEL 1,ACC 100,APO_DIST 5,APO_FAC 50.0,ORI_TYP #VAR,CIRC_TYP #BASE,JERK_FAC 50.0}
DECL FDAT FP84={TOOL_NO 2,BASE_NO 10,IPO_FRAME #BASE,POINT2[] " ",TQ_STATE FALSE}
DECL E6POS XP84={X -69.520,Y 128.040,Z -46.030,A 0.000,B -3.810,C -7.040}
DECL LDAT LCPDATP85={VEL 1,ACC 100,APO_DIST 5,APO_FAC 50.0,ORI_TYP #VAR,CIRC_TYP #BASE,JERK_FAC 50.0}
DECL FDAT FP85={TOOL_NO 2,BASE_NO 10,IPO_FRAME #BASE,POINT2[] " ",TQ_STATE FALSE}
DECL E6POS XP85={X -66.560,Y 122.590,Z -44.620,A 0.000,B -8.300,C -15.580}
DECL LDAT LCPDATC86={VEL 0.1,ACC 100,APO_DIST 5,APO_FAC 50.0,ORI_TYP #VAR,CIRC_TYP #BASE,JERK_FAC 50.0}
DECL FDAT FC86={TOOL_NO 2,BASE_NO 10,IPO_FRAME #BASE,POINT2[] " ",TQ_STATE FALSE}
DECL E6POS XCAux86={X -53.380,Y 128.870,Z -44.620,A 0.000,B -6.640,C -16.330}
DECL E6POS XCDes86={X 53.380,Y 128.870,Z -44.620,A 0.000,B 6.640,C -16.330}
DECL LDAT LCPDATP87={VEL 1,ACC 100,APO_DIST 5,APO_FAC 50.0,ORI_TYP #VAR,CIRC_TYP #BASE,JERK_FAC 50.0}
DECL FDAT FP87={TOOL_NO 2,BASE_NO 10,IPO_FRAME #BASE,POINT2[] " ",TQ_STATE FALSE}
DECL E6POS XP87={X 66.560,Y 122.590,Z -44.620,A 0.000,B 8.300,C -15.580}
DECL LDAT LCPDATP88={VEL 1,ACC 100,APO_DIST 5,APO_FAC 50.0,ORI_TYP #VAR,CIRC_TYP #BASE,JERK_FAC 50.0}
DECL FDAT FP88={TOOL_NO 2,BASE_NO 10,IPO_FRAME #BASE,POINT2[] " ",TQ_STATE FALSE}
DECL E6POS XP88={X 63.750,Y 117.420,Z -42.190,A -0.000,B 12.600,C -24.300}
DECL LDAT LCPDATC89={VEL 0.1,ACC 100,APO_DIST 5,APO_FAC 50.0,ORI_TYP #VAR,CIRC_TYP #BASE,JERK_FAC 50.0}
DECL FDAT FC89={TOOL_NO 2,BASE_NO 10,IPO_FRAME #BASE,POINT2[] " ",TQ_STATE FALSE}
DECL E6POS XCAux89={X 51.130,Y 123.440,Z -42.190,A 0.000,B 10.070,C -25.390}
DECL E6POS XCDes89={X -51.130,Y 123.440,Z -42.190,A 0.000,B -10.070,C -25.390}
DECL LDAT LCPDATP90={VEL 1,ACC 100,APO_DIST 5,APO_FAC 50.0,ORI_TYP #VAR,CIRC_TYP #BASE,JERK_FAC 50.0}
DECL FDAT FP90={TOOL_NO 2,BASE_NO 10,IPO_FRAME #BASE,POINT2[] " ",TQ_STATE FALSE}
DECL E6POS XP90={X -63.750,Y 117.420,Z -42.190,A 0.000,B -12.600,C -24.300}
DECL LDAT LCPDATP91={VEL 1,ACC 100,APO_DIST 5,APO_FAC 50.0,ORI_TYP #VAR,CIRC_TYP #BASE,JERK_FAC 50.0}
DECL FDAT FP91={TOOL_NO 2,BASE_NO 10,IPO_FRAME #BASE,POINT2[] " ",TQ_STATE FALSE}
DECL E6POS XP91={X -61.180,Y 112.670,Z -38.820,A 0.000,B -16.600,C -33.310}
DECL LDAT LCPDATC92={VEL 0.1,ACC 100,APO_DIST 5,APO_FAC 50.0,ORI_TYP #VAR,CIRC_TYP #BASE,JERK_FAC 50.0}
DECL FDAT FC92={TOOL_NO 2,BASE_NO 10,IPO_FRAME #BASE,POINT2[] " ",TQ_STATE FALSE}
DECL E6POS XCAux92={X -49.060,Y 118.450,Z -38.820,A 0.000,B -13.250,C -34.640}
DECL E6POS XCDes92={X 49.060,Y 118.450,Z -38.820,A 0.000,B 13.250,C -34.640}
DECL LDAT LCPDATP93={VEL 1,ACC 100,APO_DIST 5,APO_FAC 50.0,ORI_TYP #VAR,CIRC_TYP #BASE,JERK_FAC 50.0}
DECL FDAT FP93={TOOL_NO 2,BASE_NO 10,IPO_FRAME #BASE,POINT2[] " ",TQ_STATE FALSE}
DECL E6POS XP93={X 61.180,Y 112.670,Z -38.820,A 0.000,B 16.600,C -33.310}
DECL LDAT LCPDATP94={VEL 1,ACC 100,APO_DIST 5,APO_FAC 50.0,ORI_TYP #VAR,CIRC_TYP #BASE,JERK_FAC 50.0}
DECL FDAT FP94={TOOL_NO 2,BASE_NO 10,IPO_FRAME #BASE,POINT2[] " ",TQ_STATE FALSE}
DECL E6POS XP94={X 60.260,Y 110.980,Z -37.800,A -0.000,B 17.860,C -36.410}
DECL LDAT LCPDATC95={VEL 0.1,ACC 100,APO_DIST 5,APO_FAC 50.0,ORI_TYP #VAR,CIRC_TYP #BASE,JERK_FAC 50.0}
DECL FDAT FC95={TOOL_NO 2,BASE_NO 10,IPO_FRAME #BASE,POINT2[] " ",TQ_STATE FALSE}
DECL E6POS XCAux95={X 48.330,Y 116.670,Z -37.800,A 0.000,B 14.240,C -37.780}
DECL E6POS XCDes95={X -48.330,Y 116.670,Z -37.800,A -0.000,B -14.240,C -37.780}
DECL LDAT LCPDATP96={VEL 1,ACC 100,APO_DIST 5,APO_FAC 50.0,ORI_TYP #VAR,CIRC_TYP #BASE,JERK_FAC 50.0}
DECL FDAT FP96={TOOL_NO 2,BASE_NO 10,IPO_FRAME #BASE,POINT2[] " ",TQ_STATE FALSE}
DECL E6POS XP96={X -60.260,Y 110.980,Z -37.800,A -0.000,B -17.860,C -36.410}
DECL LDAT LCPDATP97={VEL 1,ACC 100,APO_DIST 5,APO_FAC 50.0,ORI_TYP #VAR,CIRC_TYP #BASE,JERK_FAC 50.0}
DECL FDAT FP97={TOOL_NO 2,BASE_NO 10,IPO_FRAME #BASE,POINT2[] " ",TQ_STATE FALSE}
DECL E6POS XP97={X -62.860,Y 115.770,Z -41.620,A 0.000,B -13.830,C -26.970}
DECL LDAT LCPDATC98={VEL 0.1,ACC 100,APO_DIST 5,APO_FAC 50.0,ORI_TYP #VAR,CIRC_TYP #BASE,JERK_FAC 50.0}
DECL FDAT FC98={TOOL_NO 2,BASE_NO 10,IPO_FRAME #BASE,POINT2[] " ",TQ_STATE FALSE}
DECL E6POS XCAux98={X -50.410,Y 121.700,Z -41.620,A -0.000,B -11.060,C -28.140}
DECL E6POS XCDes98={X 50.410,Y 121.700,Z -41.620,A -0.000,B 11.060,C -28.140}
DECL LDAT LCPDATP99={VEL 1,ACC 100,APO_DIST 5,APO_FAC 50.0,ORI_TYP #VAR,CIRC_TYP #BASE,JERK_FAC 50.0}
DECL FDAT FP99={TOOL_NO 2,BASE_NO 10,IPO_FRAME #BASE,POINT2[] " ",TQ_STATE FALSE}
DECL E6POS XP99={X 62.860,Y 115.770,Z -41.620,A 0.000,B 13.830,C -26.970}
DECL LDAT LCPDATP100={VEL 1,ACC 100,APO_DIST 5,APO_FAC 50.0,ORI_TYP #VAR,CIRC_TYP #BASE,JERK_FAC 50.0}
DECL FDAT FP100={TOOL_NO 2,BASE_NO 10,IPO_FRAME #BASE,POINT2[] " ",TQ_STATE FALSE}
DECL E6POS XP100={X 65.730,Y 121.060,Z -44.450,A 0.000,B 9.460,C -17.870}
DECL LDAT LCPDATC101={VEL 0.1,ACC 100,APO_DIST 5,APO_FAC 50.0,ORI_TYP #VAR,CIRC_TYP #BASE,JERK_FAC 50.0}
DECL FDAT FC101={TOOL_NO 2,BASE_NO 10,IPO_FRAME #BASE,POINT2[] " ",TQ_STATE FALSE}
DECL E6POS XCAux101={X 52.720,Y 127.270,Z -44.450,A -0.000,B 7.570,C -18.720}
DECL E6POS XCDes101={X -52.720,Y 127.270,Z -44.450,A -0.000,B -7.570,C -18.720}
DECL LDAT LCPDATP102={VEL 1,ACC 100,APO_DIST 5,APO_FAC 50.0,ORI_TYP #VAR,CIRC_TYP #BASE,JERK_FAC 50.0}
DECL FDAT FP102={TOOL_NO 2,BASE_NO 10,IPO_FRAME #BASE,POINT2[] " ",TQ_STATE FALSE}
DECL E6POS XP102={X -65.730,Y 121.060,Z -44.450,A -0.000,B -9.460,C -17.870}
DECL LDAT LCPDATP103={VEL 1,ACC 100,APO_DIST 5,APO_FAC 50.0,ORI_TYP #VAR,CIRC_TYP #BASE,JERK_FAC 50.0}
DECL FDAT FP103={TOOL_NO 2,BASE_NO 10,IPO_FRAME #BASE,POINT2[] " ",TQ_STATE FALSE}
DECL E6POS XP103={X -68.800,Y 126.710,Z -46.190,A 0.000,B -4.850,C -9.000}
DECL LDAT LCPDATC104={VEL 0.1,ACC 100,APO_DIST 5,APO_FAC 50.0,ORI_TYP #VAR,CIRC_TYP #BASE,JERK_FAC 50.0}
DECL FDAT FC104={TOOL_NO 2,BASE_NO 10,IPO_FRAME #BASE,POINT2[] " ",TQ_STATE FALSE}
DECL E6POS XCAux104={X -55.170,Y 133.200,Z -46.190,A 0.000,B -3.890,C -9.450}
DECL E6POS XCDes104={X 55.170,Y 133.200,Z -46.190,A 0.000,B 3.890,C -9.450}
DECL LDAT LCPDATP105={VEL 1,ACC 100,APO_DIST 5,APO_FAC 50.0,ORI_TYP #VAR,CIRC_TYP #BASE,JERK_FAC 50.0}
DECL FDAT FP105={TOOL_NO 2,BASE_NO 10,IPO_FRAME #BASE,POINT2[] " ",TQ_STATE FALSE}
DECL E6POS XP105={X 68.800,Y 126.710,Z -46.190,A 0.000,B 4.850,C -9.000}
DECL LDAT LCPDATP106={VEL 1,ACC 100,APO_DIST 5,APO_FAC 50.0,ORI_TYP #VAR,CIRC_TYP #BASE,JERK_FAC 50.0}
DECL FDAT FP106={TOOL_NO 2,BASE_NO 10,IPO_FRAME #BASE,POINT2[] " ",TQ_STATE FALSE}
DECL E6POS XP106={X 71.960,Y 132.530,Z -46.800,A -0.000,B 0.140,C -0.250}
DECL LDAT LCPDATC107={VEL 0.1,ACC 100,APO_DIST 5,APO_FAC 50.0,ORI_TYP #VAR,CIRC_TYP #BASE,JERK_FAC 50.0}
DECL FDAT FC107={TOOL_NO 2,BASE_NO 10,IPO_FRAME #BASE,POINT2[] " ",TQ_STATE FALSE}
DECL E6POS XCAux107={X 57.710,Y 139.330,Z -46.800,A -0.000,B 0.110,C -0.270}
DECL E6POS XCDes107={X -57.710,Y 139.330,Z -46.800,A 0.000,B -0.110,C -0.270}
DECL LDAT LCPDATP108={VEL 1,ACC 100,APO_DIST 5,APO_FAC 50.0,ORI_TYP #VAR,CIRC_TYP #BASE,JERK_FAC 50.0}
DECL FDAT FP108={TOOL_NO 2,BASE_NO 10,IPO_FRAME #BASE,POINT2[] " ",TQ_STATE FALSE}
DECL E6POS XP108={X -71.960,Y 132.530,Z -46.800,A -0.000,B -0.140,C -0.250}
DECL LDAT LCPDATP109={VEL 1,ACC 100,APO_DIST 5,APO_FAC 50.0,ORI_TYP #VAR,CIRC_TYP #BASE,JERK_FAC 50.0}
DECL FDAT FP109={TOOL_NO 2,BASE_NO 10,IPO_FRAME #BASE,POINT2[] " ",TQ_STATE FALSE}
DECL E6POS XP109={X -71.120,Y 130.990,Z -46.800,A 0.000,B 0.000,C -0.000}
DECL LDAT LCPDATC110={VEL 0.1,ACC 100,APO_DIST 5,APO_FAC 50.0,ORI_TYP #VAR,CIRC_TYP #BASE,JERK_FAC 50.0}
DECL FDAT FC110={TOOL_NO 2,BASE_NO 10,IPO_FRAME #BASE,POINT2[] " ",TQ_STATE FALSE}
DECL E6POS XCAux110={X -57.040,Y 137.710,Z -46.800,A 0.000,B 0.000,C -0.000}
DECL E6POS XCDes110={X 57.040,Y 137.710,Z -46.800,A 0.000,B 0.000,C -0.000}
DECL LDAT LCPDATP111={VEL 1,ACC 100,APO_DIST 5,APO_FAC 50.0,ORI_TYP #VAR,CIRC_TYP #BASE,JERK_FAC 50.0}
DECL FDAT FP111={TOOL_NO 2,BASE_NO 10,IPO_FRAME #BASE,POINT2[] " ",TQ_STATE FALSE}
DECL E6POS XP111={X 71.120,Y 130.990,Z -46.800,A 0.000,B 0.000,C -0.000}
DECL LDAT LCPDATP112={VEL 1,ACC 100,APO_DIST 5,APO_FAC 50.0,ORI_TYP #VAR,CIRC_TYP #BASE,JERK_FAC 50.0}
DECL FDAT FP112={TOOL_NO 2,BASE_NO 10,IPO_FRAME #BASE,POINT2[] " ",TQ_STATE FALSE}
DECL E6POS XP112={X 70.170,Y 129.240,Z -46.800,A 0.000,B 0.000,C -0.000}
DECL LDAT LCPDATC113={VEL 0.1,ACC 100,APO_DIST 5,APO_FAC 50.0,ORI_TYP #VAR,CIRC_TYP #BASE,JERK_FAC 50.0}
DECL FDAT FC113={TOOL_NO 2,BASE_NO 10,IPO_FRAME #BASE,POINT2[] " ",TQ_STATE FALSE}
DECL E6POS XCAux113={X 56.280,Y 135.860,Z -46.800,A 0.000,B 0.000,C -0.000}
DECL E6POS XCDes113={X -56.280,Y 135.860,Z -46.800,A 0.000,B 0.000,C -0.000}
DECL LDAT LCPDATP114={VEL 1,ACC 100,APO_DIST 5,APO_FAC 50.0,ORI_TYP #VAR,CIRC_TYP #BASE,JERK_FAC 50.0}
DECL FDAT FP114={TOOL_NO 2,BASE_NO 10,IPO_FRAME #BASE,POINT2[] " ",TQ_STATE FALSE}
DECL E6POS XP114={X -70.170,Y 129.240,Z -46.800,A 0.000,B 0.000,C -0.000}
DECL LDAT LCPDATP115={VEL 1,ACC 100,APO_DIST 5,APO_FAC 50.0,ORI_TYP #VAR,CIRC_TYP #BASE,JERK_FAC 50.0}
DECL FDAT FP115={TOOL_NO 2,BASE_NO 10,IPO_FRAME #BASE,POINT2[] " ",TQ_STATE FALSE}
DECL E6POS XP115={X -69.220,Y 127.480,Z -46.800,A 0.000,B 0.000,C -0.000}
DECL LDAT LCPDATC116={VEL 0.1,ACC 100,APO_DIST 5,APO_FAC 50.0,ORI_TYP #VAR,CIRC_TYP #BASE,JERK_FAC 50.0}
DECL FDAT FC116={TOOL_NO 2,BASE_NO 10,IPO_FRAME #BASE,POINT2[] " ",TQ_STATE FALSE}
DECL E6POS XCAux116={X -55.510,Y 134.020,Z -46.800,A 0.000,B 0.000,C -0.000}
DECL E6POS XCDes116={X 55.510,Y 134.020,Z -46.800,A 0.000,B 0.000,C -0.000}
DECL LDAT LCPDATP117={VEL 1,ACC 100,APO_DIST 5,APO_FAC 50.0,ORI_TYP #VAR,CIRC_TYP #BASE,JERK_FAC 50.0}
DECL FDAT FP117={TOOL_NO 2,BASE_NO 10,IPO_FRAME #BASE,POINT2[] " ",TQ_STATE FALSE}
DECL E6POS XP117={X 69.220,Y 127.480,Z -46.800,A 0.000,B 0.000,C -0.000}
DECL LDAT LCPDATP118={VEL 1,ACC 100,APO_DIST 5,APO_FAC 50.0,ORI_TYP #VAR,CIRC_TYP #BASE,JERK_FAC 50.0}
DECL FDAT FP118={TOOL_NO 2,BASE_NO 10,IPO_FRAME #BASE,POINT2[] " ",TQ_STATE FALSE}
DECL E6POS XP118={X 68.260,Y 125.720,Z -46.800,A 0.000,B 0.000,C -0.000}
DECL LDAT LCPDATC119={VEL 0.1,ACC 100,APO_DIST 5,APO_FAC 50.0,ORI_TYP #VAR,CIRC_TYP #BASE,JERK_FAC 50.0}
DECL FDAT FC119={TOOL_NO 2,BASE_NO 10,IPO_FRAME #BASE,POINT2[] " ",TQ_STATE FALSE}
DECL E6POS XCAux119={X 54.750,Y 132.170,Z -46.800,A 0.000,B 0.000,C -0.000}
DECL E6POS XCDes119={X -54.750,Y 132.170,Z -46.800,A 0.000,B 0.000,C -0.000}
DECL LDAT LCPDATP120={VEL 1,ACC 100,APO_DIST 5,APO_FAC 50.0,ORI_TYP #VAR,CIRC_TYP #BASE,JERK_FAC 50.0}
DECL FDAT FP120={TOOL_NO 2,BASE_NO 10,IPO_FRAME #BASE,POINT2[] " ",TQ_STATE FALSE}
DECL E6POS XP120={X -68.260,Y 125.720,Z -46.800,A 0.000,B 0.000,C -0.000}
DECL LDAT LCPDATP121={VEL 1,ACC 100,APO_DIST 5,APO_FAC 50.0,ORI_TYP #VAR,CIRC_TYP #BASE,JERK_FAC 50.0}
DECL FDAT FP121={TOOL_NO 2,BASE_NO 10,IPO_FRAME #BASE,POINT2[] " ",TQ_STATE FALSE}
DECL E6POS XP121={X -67.310,Y 123.960,Z -46.800,A 0.000,B 0.000,C -0.000}
DECL LDAT LCPDATC122={VEL 0.1,ACC 100,APO_DIST 5,APO_FAC 50.0,ORI_TYP #VAR,CIRC_TYP #BASE,JERK_FAC 50.0}
DECL FDAT FC122={TOOL_NO 2,BASE_NO 10,IPO_FRAME #BASE,POINT2[] " ",TQ_STATE FALSE}
DECL E6POS XCAux122={X -53.980,Y 130.320,Z -46.800,A 0.000,B 0.000,C -0.000}
DECL E6POS XCDes122={X 53.980,Y 130.320,Z -46.800,A 0.000,B 0.000,C -0.000}
DECL LDAT LCPDATP123={VEL 1,ACC 100,APO_DIST 5,APO_FAC 50.0,ORI_TYP #VAR,CIRC_TYP #BASE,JERK_FAC 50.0}
DECL FDAT FP123={TOOL_NO 2,BASE_NO 10,IPO_FRAME #BASE,POINT2[] " ",TQ_STATE FALSE}
DECL E6POS XP123={X 67.310,Y 123.960,Z -46.800,A 0.000,B 0.000,C -0.000}
DECL LDAT LCPDATP124={VEL 1,ACC 100,APO_DIST 5,APO_FAC 50.0,ORI_TYP #VAR,CIRC_TYP #BASE,JERK_FAC 50.0}
DECL FDAT FP124={TOOL_NO 2,BASE_NO 10,IPO_FRAME #BASE,POINT2[] " ",TQ_STATE FALSE}
DECL E6POS XP124={X 66.350,Y 122.210,Z -46.800,A 0.000,B 0.000,C -0.000}
DECL LDAT LCPDATC125={VEL 0.1,ACC 100,APO_DIST 5,APO_FAC 50.0,ORI_TYP #VAR,CIRC_TYP #BASE,JERK_FAC 50.0}
DECL FDAT FC125={TOOL_NO 2,BASE_NO 10,IPO_FRAME #BASE,POINT2[] " ",TQ_STATE FALSE}
DECL E6POS XCAux125={X 53.220,Y 128.470,Z -46.800,A 0.000,B 0.000,C -0.000}
DECL E6POS XCDes125={X -53.220,Y 128.470,Z -46.800,A 0.000,B 0.000,C -0.000}
DECL LDAT LCPDATP126={VEL 1,ACC 100,APO_DIST 5,APO_FAC 50.0,ORI_TYP #VAR,CIRC_TYP #BASE,JERK_FAC 50.0}
DECL FDAT FP126={TOOL_NO 2,BASE_NO 10,IPO_FRAME #BASE,POINT2[] " ",TQ_STATE FALSE}
DECL E6POS XP126={X -66.350,Y 122.210,Z -46.800,A 0.000,B 0.000,C -0.000}
DECL LDAT LCPDATP127={VEL 1,ACC 100,APO_DIST 5,APO_FAC 50.0,ORI_TYP #VAR,CIRC_TYP #BASE,JERK_FAC 50.0}
DECL FDAT FP127={TOOL_NO 2,BASE_NO 10,IPO_FRAME #BASE,POINT2[] " ",TQ_STATE FALSE}
DECL E6POS XP127={X -69.410,Y 127.840,Z -46.250,A 0.000,B 4.600,C 8.530}
DECL LDAT LCPDATC128={VEL 0.1,ACC 100,APO_DIST 5,APO_FAC 50.0,ORI_TYP #VAR,CIRC_TYP #BASE,JERK_FAC 50.0}
DECL FDAT FC128={TOOL_NO 2,BASE_NO 10,IPO_FRAME #BASE,POINT2[] " ",TQ_STATE FALSE}
DECL E6POS XCAux128={X -55.670,Y 134.400,Z -46.250,A 0.000,B 3.690,C 8.960}
DECL E6POS XCDes128={X 55.670,Y 134.400,Z -46.250,A 0.000,B -3.690,C 8.960}
DECL LDAT LCPDATP129={VEL 1,ACC 100,APO_DIST 5,APO_FAC 50.0,ORI_TYP #VAR,CIRC_TYP #BASE,JERK_FAC 50.0}
DECL FDAT FP129={TOOL_NO 2,BASE_NO 10,IPO_FRAME #BASE,POINT2[] " ",TQ_STATE FALSE}
DECL E6POS XP129={X 69.410,Y 127.840,Z -46.250,A 0.000,B -4.600,C 8.530}
DECL LDAT LCPDATP130={VEL 1,ACC 100,APO_DIST 5,APO_FAC 50.0,ORI_TYP #VAR,CIRC_TYP #BASE,JERK_FAC 50.0}
DECL FDAT FP130={TOOL_NO 2,BASE_NO 10,IPO_FRAME #BASE,POINT2[] " ",TQ_STATE FALSE}
DECL E6POS XP130={X 72.480,Y 133.500,Z -44.570,A 0.000,B -9.220,C 17.390}
DECL LDAT LCPDATC131={VEL 0.1,ACC 100,APO_DIST 5,APO_FAC 50.0,ORI_TYP #VAR,CIRC_TYP #BASE,JERK_FAC 50.0}
DECL FDAT FC131={TOOL_NO 2,BASE_NO 10,IPO_FRAME #BASE,POINT2[] " ",TQ_STATE FALSE}
DECL E6POS XCAux131={X 58.130,Y 140.350,Z -44.570,A 0.000,B -7.380,C 18.220}
DECL E6POS XCDes131={X -58.130,Y 140.350,Z -44.570,A 0.000,B 7.380,C 18.220}
DECL LDAT LCPDATP132={VEL 1,ACC 100,APO_DIST 5,APO_FAC 50.0,ORI_TYP #VAR,CIRC_TYP #BASE,JERK_FAC 50.0}
DECL FDAT FP132={TOOL_NO 2,BASE_NO 10,IPO_FRAME #BASE,POINT2[] " ",TQ_STATE FALSE}
DECL E6POS XP132={X -72.480,Y 133.500,Z -44.570,A 0.000,B 9.220,C 17.390}
DECL LDAT LCPDATP133={VEL 1,ACC 100,APO_DIST 5,APO_FAC 50.0,ORI_TYP #VAR,CIRC_TYP #BASE,JERK_FAC 50.0}
DECL FDAT FP133={TOOL_NO 2,BASE_NO 10,IPO_FRAME #BASE,POINT2[] " ",TQ_STATE FALSE}
DECL E6POS XP133={X -75.370,Y 138.820,Z -41.800,A 0.000,B 13.610,C 26.480}
DECL LDAT LCPDATC134={VEL 0.1,ACC 100,APO_DIST 5,APO_FAC 50.0,ORI_TYP #VAR,CIRC_TYP #BASE,JERK_FAC 50.0}
DECL FDAT FC134={TOOL_NO 2,BASE_NO 10,IPO_FRAME #BASE,POINT2[] " ",TQ_STATE FALSE}
DECL E6POS XCAux134={X -60.450,Y 145.940,Z -41.800,A 0.000,B 10.880,C 27.640}
DECL E6POS XCDes134={X 60.450,Y 145.940,Z -41.800,A 0.000,B -10.880,C 27.640}
DECL LDAT LCPDATP135={VEL 1,ACC 100,APO_DIST 5,APO_FAC 50.0,ORI_TYP #VAR,CIRC_TYP #BASE,JERK_FAC 50.0}
DECL FDAT FP135={TOOL_NO 2,BASE_NO 10,IPO_FRAME #BASE,POINT2[] " ",TQ_STATE FALSE}
DECL E6POS XP135={X 75.370,Y 138.820,Z -41.800,A 0.000,B -13.610,C 26.480}
DECL LDAT LCPDATP136={VEL 1,ACC 100,APO_DIST 5,APO_FAC 50.0,ORI_TYP #VAR,CIRC_TYP #BASE,JERK_FAC 50.0}
DECL FDAT FP136={TOOL_NO 2,BASE_NO 10,IPO_FRAME #BASE,POINT2[] " ",TQ_STATE FALSE}
DECL E6POS XP136={X 77.990,Y 143.640,Z -38.030,A 0.000,B -17.660,C 35.890}
DECL LDAT LCPDATC137={VEL 0.1,ACC 100,APO_DIST 5,APO_FAC 50.0,ORI_TYP #VAR,CIRC_TYP #BASE,JERK_FAC 50.0}
DECL FDAT FC137={TOOL_NO 2,BASE_NO 10,IPO_FRAME #BASE,POINT2[] " ",TQ_STATE FALSE}
DECL E6POS XCAux137={X 62.550,Y 151.000,Z -38.030,A 0.000,B -14.080,C 37.260}
DECL E6POS XCDes137={X -62.550,Y 151.000,Z -38.030,A 0.000,B 14.080,C 37.260}
DECL LDAT LCPDATP138={VEL 1,ACC 100,APO_DIST 5,APO_FAC 50.0,ORI_TYP #VAR,CIRC_TYP #BASE,JERK_FAC 50.0}
DECL FDAT FP138={TOOL_NO 2,BASE_NO 10,IPO_FRAME #BASE,POINT2[] " ",TQ_STATE FALSE}
DECL E6POS XP138={X -77.990,Y 143.640,Z -38.030,A 0.000,B 17.660,C 35.890}
DECL LDAT LCPDATP139={VEL 1,ACC 100,APO_DIST 5,APO_FAC 50.0,ORI_TYP #VAR,CIRC_TYP #BASE,JERK_FAC 50.0}
DECL FDAT FP139={TOOL_NO 2,BASE_NO 10,IPO_FRAME #BASE,POINT2[] " ",TQ_STATE FALSE}
DECL E6POS XP139={X -78.240,Y 144.110,Z -38.110,A -0.000,B 17.860,C 36.410}
DECL LDAT LCPDATC140={VEL 0.1,ACC 100,APO_DIST 5,APO_FAC 50.0,ORI_TYP #VAR,CIRC_TYP #BASE,JERK_FAC 50.0}
DECL FDAT FC140={TOOL_NO 2,BASE_NO 10,IPO_FRAME #BASE,POINT2[] " ",TQ_STATE FALSE}
DECL E6POS XCAux140={X -62.750,Y 151.500,Z -38.110,A -0.000,B 14.240,C 37.780}
DECL E6POS XCDes140={X 62.750,Y 151.500,Z -38.110,A 0.000,B -14.240,C 37.780}
DECL LDAT LCPDATP141={VEL 1,ACC 100,APO_DIST 5,APO_FAC 50.0,ORI_TYP #VAR,CIRC_TYP #BASE,JERK_FAC 50.0}
DECL FDAT FP141={TOOL_NO 2,BASE_NO 10,IPO_FRAME #BASE,POINT2[] " ",TQ_STATE FALSE}
DECL E6POS XP141={X 78.240,Y 144.110,Z -38.110,A -0.000,B -17.860,C 36.410}
DECL LDAT LCPDATP142={VEL 1,ACC 100,APO_DIST 5,APO_FAC 50.0,ORI_TYP #VAR,CIRC_TYP #BASE,JERK_FAC 50.0}
DECL FDAT FP142={TOOL_NO 2,BASE_NO 10,IPO_FRAME #BASE,POINT2[] " ",TQ_STATE FALSE}
DECL E6POS XP142={X 75.520,Y 139.080,Z -42.090,A 0.000,B -13.680,C 26.640}
DECL LDAT LCPDATC143={VEL 0.1,ACC 100,APO_DIST 5,APO_FAC 50.0,ORI_TYP #VAR,CIRC_TYP #BASE,JERK_FAC 50.0}
DECL FDAT FC143={TOOL_NO 2,BASE_NO 10,IPO_FRAME #BASE,POINT2[] " ",TQ_STATE FALSE}
DECL E6POS XCAux143={X 60.560,Y 146.210,Z -42.090,A 0.000,B -10.930,C 27.800}
DECL E6POS XCDes143={X -60.560,Y 146.210,Z -42.090,A -0.000,B 10.930,C 27.800}
DECL LDAT LCPDATP144={VEL 1,ACC 100,APO_DIST 5,APO_FAC 50.0,ORI_TYP #VAR,CIRC_TYP #BASE,JERK_FAC 50.0}
DECL FDAT FP144={TOOL_NO 2,BASE_NO 10,IPO_FRAME #BASE,POINT2[] " ",TQ_STATE FALSE}
DECL E6POS XP144={X -75.520,Y 139.080,Z -42.090,A -0.000,B 13.680,C 26.640}
DECL LDAT LCPDATP145={VEL 1,ACC 100,APO_DIST 5,APO_FAC 50.0,ORI_TYP #VAR,CIRC_TYP #BASE,JERK_FAC 50.0}
DECL FDAT FP145={TOOL_NO 2,BASE_NO 10,IPO_FRAME #BASE,POINT2[] " ",TQ_STATE FALSE}
DECL E6POS XP145={X -72.490,Y 133.520,Z -44.990,A -0.000,B 9.130,C 17.220}
DECL LDAT LCPDATC146={VEL 0.1,ACC 100,APO_DIST 5,APO_FAC 50.0,ORI_TYP #VAR,CIRC_TYP #BASE,JERK_FAC 50.0}
DECL FDAT FC146={TOOL_NO 2,BASE_NO 10,IPO_FRAME #BASE,POINT2[] " ",TQ_STATE FALSE}
DECL E6POS XCAux146={X -58.140,Y 140.360,Z -44.990,A 0.000,B 7.310,C 18.050}
DECL E6POS XCDes146={X 58.140,Y 140.360,Z -44.990,A -0.000,B -7.310,C 18.050}
DECL LDAT LCPDATP147={VEL 1,ACC 100,APO_DIST 5,APO_FAC 50.0,ORI_TYP #VAR,CIRC_TYP #BASE,JERK_FAC 50.0}
DECL FDAT FP147={TOOL_NO 2,BASE_NO 10,IPO_FRAME #BASE,POINT2[] " ",TQ_STATE FALSE}
DECL E6POS XP147={X 72.490,Y 133.520,Z -44.990,A -0.000,B -9.130,C 17.220}
DECL LDAT LCPDATP148={VEL 1,ACC 100,APO_DIST 5,APO_FAC 50.0,ORI_TYP #VAR,CIRC_TYP #BASE,JERK_FAC 50.0}
DECL FDAT FP148={TOOL_NO 2,BASE_NO 10,IPO_FRAME #BASE,POINT2[] " ",TQ_STATE FALSE}
DECL E6POS XP148={X 69.270,Y 127.580,Z -46.710,A 0.000,B -4.350,C 8.050}
DECL LDAT LCPDATC149={VEL 0.1,ACC 100,APO_DIST 5,APO_FAC 50.0,ORI_TYP #VAR,CIRC_TYP #BASE,JERK_FAC 50.0}
DECL FDAT FC149={TOOL_NO 2,BASE_NO 10,IPO_FRAME #BASE,POINT2[] " ",TQ_STATE FALSE}
DECL E6POS XCAux149={X 55.560,Y 134.130,Z -46.710,A -0.000,B -3.490,C 8.460}
DECL E6POS XCDes149={X -55.560,Y 134.130,Z -46.710,A -0.000,B 3.490,C 8.460}
DECL LDAT LCPDATP150={VEL 1,ACC 100,APO_DIST 5,APO_FAC 50.0,ORI_TYP #VAR,CIRC_TYP #BASE,JERK_FAC 50.0}
DECL FDAT FP150={TOOL_NO 2,BASE_NO 10,IPO_FRAME #BASE,POINT2[] " ",TQ_STATE FALSE}
DECL E6POS XP150={X -69.270,Y 127.580,Z -46.710,A -0.000,B 4.350,C 8.050}
DECL LDAT LCPDATP151={VEL 1,ACC 100,APO_DIST 5,APO_FAC 50.0,ORI_TYP #VAR,CIRC_TYP #BASE,JERK_FAC 50.0}
DECL FDAT FP151={TOOL_NO 2,BASE_NO 10,IPO_FRAME #BASE,POINT2[] " ",TQ_STATE FALSE}
DECL E6POS XP151={X -66.430,Y 122.360,Z -47.200,A 0.000,B 0.000,C -0.000}
DECL LDAT LCPDATC152={VEL 0.1,ACC 100,APO_DIST 5,APO_FAC 50.0,ORI_TYP #VAR,CIRC_TYP #BASE,JERK_FAC 50.0}
DECL FDAT FC152={TOOL_NO 2,BASE_NO 10,IPO_FRAME #BASE,POINT2[] " ",TQ_STATE FALSE}
DECL E6POS XCAux152={X -53.280,Y 128.630,Z -47.200,A 0.000,B 0.000,C -0.000}
DECL E6POS XCDes152={X 53.280,Y 128.630,Z -47.200,A 0.000,B 0.000,C -0.000}
DECL LDAT LCPDATP153={VEL 1,ACC 100,APO_DIST 5,APO_FAC 50.0,ORI_TYP #VAR,CIRC_TYP #BASE,JERK_FAC 50.0}
DECL FDAT FP153={TOOL_NO 2,BASE_NO 10,IPO_FRAME #BASE,POINT2[] " ",TQ_STATE FALSE}
DECL E6POS XP153={X 66.430,Y 122.360,Z -47.200,A 0.000,B 0.000,C -0.000}
DECL LDAT LCPDATP154={VEL 1,ACC 100,APO_DIST 5,APO_FAC 50.0,ORI_TYP #VAR,CIRC_TYP #BASE,JERK_FAC 50.0}
DECL FDAT FP154={TOOL_NO 2,BASE_NO 10,IPO_FRAME #BASE,POINT2[] " ",TQ_STATE FALSE}
DECL E6POS XP154={X 67.390,Y 124.110,Z -47.200,A 0.000,B 0.000,C -0.000}
DECL LDAT LCPDATC155={VEL 0.1,ACC 100,APO_DIST 5,APO_FAC 50.0,ORI_TYP #VAR,CIRC_TYP #BASE,JERK_FAC 50.0}
DECL FDAT FC155={TOOL_NO 2,BASE_NO 10,IPO_FRAME #BASE,POINT2[] " ",TQ_STATE FALSE}
DECL E6POS XCAux155={X 54.050,Y 130.480,Z -47.200,A 0.000,B 0.000,C -0.000}
DECL E6POS XCDes155={X -54.050,Y 130.480,Z -47.200,A 0.000,B 0.000,C -0.000}
DECL LDAT LCPDATP156={VEL 1,ACC 100,APO_DIST 5,APO_FAC 50.0,ORI_TYP #VAR,CIRC_TYP #BASE,JERK_FAC 50.0}
DECL FDAT FP156={TOOL_NO 2,BASE_NO 10,IPO_FRAME #BASE,POINT2[] " ",TQ_STATE FALSE}
DECL E6POS XP156={X -67.390,Y 124.110,Z -47.200,A 0.000,B 0.000,C -0.000}
DECL LDAT LCPDATP157={VEL 1,ACC 100,APO_DIST 5,APO_FAC 50.0,ORI_TYP #VAR,CIRC_TYP #BASE,JERK_FAC 50.0}
DECL FDAT FP157={TOOL_NO 2,BASE_NO 10,IPO_FRAME #BASE,POINT2[] " ",TQ_STATE FALSE}
DECL E6POS XP157={X -68.340,Y 125.870,Z -47.200,A 0.000,B 0.000,C -0.000}
DECL LDAT LCPDATC158={VEL 0.1,ACC 100,APO_DIST 5,APO_FAC 50.0,ORI_TYP #VAR,CIRC_TYP #BASE,JERK_FAC 50.0}
DECL FDAT FC158={TOOL_NO 2,BASE_NO 10,IPO_FRAME #BASE,POINT2[] " ",TQ_STATE FALSE}
DECL E6POS XCAux158={X -54.810,Y 132.330,Z -47.200,A 0.000,B 0.000,C -0.000}
DECL E6POS XCDes158={X 54.810,Y 132.330,Z -47.200,A 0.000,B 0.000,C -0.000}
DECL LDAT LCPDATP159={VEL 1,ACC 100,APO_DIST 5,APO_FAC 50.0,ORI_TYP #VAR,CIRC_TYP #BASE,JERK_FAC 50.0}
DECL FDAT FP159={TOOL_NO 2,BASE_NO 10,IPO_FRAME #BASE,POINT2[] " ",TQ_STATE FALSE}
DECL E6POS XP159={X 68.340,Y 125.870,Z -47.200,A 0.000,B 0.000,C -0.000}
DECL LDAT LCPDATP160={VEL 1,ACC 100,APO_DIST 5,APO_FAC 50.0,ORI_TYP #VAR,CIRC_TYP #BASE,JERK_FAC 50.0}
DECL FDAT FP160={TOOL_NO 2,BASE_NO 10,IPO_FRAME #BASE,POINT2[] " ",TQ_STATE FALSE}
DECL E6POS XP160={X 69.300,Y 127.630,Z -47.200,A 0.000,B 0.000,C -0.000}
DECL LDAT LCPDATC161={VEL 0.1,ACC 100,APO_DIST 5,APO_FAC 50.0,ORI_TYP #VAR,CIRC_TYP #BASE,JERK_FAC 50.0}
DECL FDAT FC161={TOOL_NO 2,BASE_NO 10,IPO_FRAME #BASE,POINT2[] " ",TQ_STATE FALSE}
DECL E6POS XCAux161={X 55.580,Y 134.170,Z -47.200,A 0.000,B 0.000,C -0.000}
DECL E6POS XCDes161={X -55.580,Y 134.170,Z -47.200,A 0.000,B 0.000,C -0.000}
DECL LDAT LCPDATP162={VEL 1,ACC 100,APO_DIST 5,APO_FAC 50.0,ORI_TYP #VAR,CIRC_TYP #BASE,JERK_FAC 50.0}
DECL FDAT FP162={TOOL_NO 2,BASE_NO 10,IPO_FRAME #BASE,POINT2[] " ",TQ_STATE FALSE}
DECL E6POS XP162={X -69.300,Y 127.630,Z -47.200,A 0.000,B 0.000,C -0.000}
DECL LDAT LCPDATP163={VEL 1,ACC 100,APO_DIST 5,APO_FAC 50.0,ORI_TYP #VAR,CIRC_TYP #BASE,JERK_FAC 50.0}
DECL FDAT FP163={TOOL_NO 2,BASE_NO 10,IPO_FRAME #BASE,POINT2[] " ",TQ_STATE FALSE}
DECL E6POS XP163={X -70.250,Y 129.390,Z -47.200,A 0.000,B 0.000,C -0.000}
DECL LDAT LCPDATC164={VEL 0.1,ACC 100,APO_DIST 5,APO_FAC 50.0,ORI_TYP #VAR,CIRC_TYP #BASE,JERK_FAC 50.0}
DECL FDAT FC164={TOOL_NO 2,BASE_NO 10,IPO_FRAME #BASE,POINT2[] " ",TQ_STATE FALSE}
DECL E6POS XCAux164={X -56.340,Y 136.020,Z -47.200,A 0.000,B 0.000,C -0.000}
DECL E6POS XCDes164={X 56.340,Y 136.020,Z -47.200,A 0.000,B 0.000,C -0.000}
DECL LDAT LCPDATP165={VEL 1,ACC 100,APO_DIST 5,APO_FAC 50.0,ORI_TYP #VAR,CIRC_TYP #BASE,JERK_FAC 50.0}
DECL FDAT FP165={TOOL_NO 2,BASE_NO 10,IPO_FRAME #BASE,POINT2[] " ",TQ_STATE FALSE}
DECL E6POS XP165={X 70.250,Y 129.390,Z -47.200,A 0.000,B 0.000,C -0.000}
DECL LDAT LCPDATP166={VEL 1,ACC 100,APO_DIST 5,APO_FAC 50.0,ORI_TYP #VAR,CIRC_TYP #BASE,JERK_FAC 50.0}
DECL FDAT FP166={TOOL_NO 2,BASE_NO 10,IPO_FRAME #BASE,POINT2[] " ",TQ_STATE FALSE}
DECL E6POS XP166={X 71.210,Y 131.140,Z -47.200,A 0.000,B 0.000,C -0.000}
DECL LDAT LCPDATC167={VEL 0.1,ACC 100,APO_DIST 5,APO_FAC 50.0,ORI_TYP #VAR,CIRC_TYP #BASE,JERK_FAC 50.0}
DECL FDAT FC167={TOOL_NO 2,BASE_NO 10,IPO_FRAME #BASE,POINT2[] " ",TQ_STATE FALSE}
DECL E6POS XCAux167={X 57.110,Y 137.870,Z -47.200,A 0.000,B 0.000,C -0.000}
DECL E6POS XCDes167={X -57.110,Y 137.870,Z -47.200,A 0.000,B 0.000,C -0.000}
DECL LDAT LCPDATP168={VEL 1,ACC 100,APO_DIST 5,APO_FAC 50.0,ORI_TYP #VAR,CIRC_TYP #BASE,JERK_FAC 50.0}
DECL FDAT FP168={TOOL_NO 2,BASE_NO 10,IPO_FRAME #BASE,POINT2[] " ",TQ_STATE FALSE}
DECL E6POS XP168={X -71.210,Y 131.140,Z -47.200,A 0.000,B 0.000,C -0.000}
DECL LDAT LCPDATP169={VEL 1,ACC 100,APO_DIST 5,APO_FAC 50.0,ORI_TYP #VAR,CIRC_TYP #BASE,JERK_FAC 50.0}
DECL FDAT FP169={TOOL_NO 2,BASE_NO 10,IPO_FRAME #BASE,POINT2[] " ",TQ_STATE FALSE}
DECL E6POS XP169={X -71.670,Y 132.000,Z -47.190,A 0.000,B -0.560,C -1.030}
DECL LDAT LCPDATC170={VEL 0.1,ACC 100,APO_DIST 5,APO_FAC 50.0,ORI_TYP #VAR,CIRC_TYP #BASE,JERK_FAC 50.0}
DECL FDAT FC170={TOOL_NO 2,BASE_NO 10,IPO_FRAME #BASE,POINT2[] " ",TQ_STATE FALSE}
DECL E6POS XCAux170={X -57.480,Y 138.770,Z -47.190,A 0.000,B -0.450,C -1.090}
DECL E6POS XCDes170={X 57.480,Y 138.770,Z -47.190,A 0.000,B 0.450,C -1.090}
DECL LDAT LCPDATP171={VEL 1,ACC 100,APO_DIST 5,APO_FAC 50.0,ORI_TYP #VAR,CIRC_TYP #BASE,JERK_FAC 50.0}
DECL FDAT FP171={TOOL_NO 2,BASE_NO 10,IPO_FRAME #BASE,POINT2[] " ",TQ_STATE FALSE}
DECL E6POS XP171={X 71.670,Y 132.000,Z -47.190,A -0.000,B 0.560,C -1.030}
DECL LDAT LCPDATP172={VEL 1,ACC 100,APO_DIST 5,APO_FAC 50.0,ORI_TYP #VAR,CIRC_TYP #BASE,JERK_FAC 50.0}
DECL FDAT FP172={TOOL_NO 2,BASE_NO 10,IPO_FRAME #BASE,POINT2[] " ",TQ_STATE FALSE}
DECL E6POS XP172={X 68.370,Y 125.920,Z -46.430,A 0.000,B 5.440,C -10.100}
DECL LDAT LCPDATC173={VEL 0.1,ACC 100,APO_DIST 5,APO_FAC 50.0,ORI_TYP #VAR,CIRC_TYP #BASE,JERK_FAC 50.0}
DECL FDAT FC173={TOOL_NO 2,BASE_NO 10,IPO_FRAME #BASE,POINT2[] " ",TQ_STATE FALSE}
DECL E6POS XCAux173={X 54.830,Y 132.370,Z -46.430,A -0.000,B 4.360,C -10.610}
DECL E6POS XCDes173={X -54.830,Y 132.370,Z -46.430,A 0.000,B -4.360,C -10.610}
DECL LDAT LCPDATP174={VEL 1,ACC 100,APO_DIST 5,APO_FAC 50.0,ORI_TYP #VAR,CIRC_TYP #BASE,JERK_FAC 50.0}
DECL FDAT FP174={TOOL_NO 2,BASE_NO 10,IPO_FRAME #BASE,POINT2[] " ",TQ_STATE FALSE}
DECL E6POS XP174={X -68.370,Y 125.920,Z -46.430,A 0.000,B -5.440,C -10.100}
DECL LDAT LCPDATP175={VEL 1,ACC 100,APO_DIST 5,APO_FAC 50.0,ORI_TYP #VAR,CIRC_TYP #BASE,JERK_FAC 50.0}
DECL FDAT FP175={TOOL_NO 2,BASE_NO 10,IPO_FRAME #BASE,POINT2[] " ",TQ_STATE FALSE}
DECL E6POS XP175={X -65.180,Y 120.050,Z -44.430,A 0.000,B -10.180,C -19.320}
DECL LDAT LCPDATC176={VEL 0.1,ACC 100,APO_DIST 5,APO_FAC 50.0,ORI_TYP #VAR,CIRC_TYP #BASE,JERK_FAC 50.0}
DECL FDAT FC176={TOOL_NO 2,BASE_NO 10,IPO_FRAME #BASE,POINT2[] " ",TQ_STATE FALSE}
DECL E6POS XCAux176={X -52.280,Y 126.210,Z -44.430,A -0.000,B -8.150,C -20.230}
DECL E6POS XCDes176={X 52.280,Y 126.210,Z -44.430,A 0.000,B 8.150,C -20.230}
DECL LDAT LCPDATP177={VEL 1,ACC 100,APO_DIST 5,APO_FAC 50.0,ORI_TYP #VAR,CIRC_TYP #BASE,JERK_FAC 50.0}
DECL FDAT FP177={TOOL_NO 2,BASE_NO 10,IPO_FRAME #BASE,POINT2[] " ",TQ_STATE FALSE}
DECL E6POS XP177={X 65.180,Y 120.050,Z -44.430,A 0.000,B 10.180,C -19.320}
DECL LDAT LCPDATP178={VEL 1,ACC 100,APO_DIST 5,APO_FAC 50.0,ORI_TYP #VAR,CIRC_TYP #BASE,JERK_FAC 50.0}
DECL FDAT FP178={TOOL_NO 2,BASE_NO 10,IPO_FRAME #BASE,POINT2[] " ",TQ_STATE FALSE}
DECL E6POS XP178={X 62.220,Y 114.590,Z -41.280,A 0.000,B 14.660,C -28.800}
DECL LDAT LCPDATC179={VEL 0.1,ACC 100,APO_DIST 5,APO_FAC 50.0,ORI_TYP #VAR,CIRC_TYP #BASE,JERK_FAC 50.0}
DECL FDAT FC179={TOOL_NO 2,BASE_NO 10,IPO_FRAME #BASE,POINT2[] " ",TQ_STATE FALSE}
DECL E6POS XCAux179={X 49.900,Y 120.470,Z -41.280,A 0.000,B 11.710,C -30.030}
DECL E6POS XCDes179={X -49.900,Y 120.470,Z -41.280,A 0.000,B -11.710,C -30.030}
DECL LDAT LCPDATP180={VEL 1,ACC 100,APO_DIST 5,APO_FAC 50.0,ORI_TYP #VAR,CIRC_TYP #BASE,JERK_FAC 50.0}
DECL FDAT FP180={TOOL_NO 2,BASE_NO 10,IPO_FRAME #BASE,POINT2[] " ",TQ_STATE FALSE}
DECL E6POS XP180={X -62.220,Y 114.590,Z -41.280,A 0.000,B -14.660,C -28.800}
DECL LDAT LCPDATP181={VEL 1,ACC 100,APO_DIST 5,APO_FAC 50.0,ORI_TYP #VAR,CIRC_TYP #BASE,JERK_FAC 50.0}
DECL FDAT FP181={TOOL_NO 2,BASE_NO 10,IPO_FRAME #BASE,POINT2[] " ",TQ_STATE FALSE}
DECL E6POS XP181={X -59.570,Y 109.710,Z -37.080,A 0.000,B -18.740,C -38.660}
DECL LDAT LCPDATC182={VEL 0.1,ACC 100,APO_DIST 5,APO_FAC 50.0,ORI_TYP #VAR,CIRC_TYP #BASE,JERK_FAC 50.0}
DECL FDAT FC182={TOOL_NO 2,BASE_NO 10,IPO_FRAME #BASE,POINT2[] " ",TQ_STATE FALSE}
DECL E6POS XCAux182={X -47.770,Y 115.340,Z -37.080,A 0.000,B -14.930,C -40.070}
DECL E6POS XCDes182={X 47.770,Y 115.340,Z -37.080,A -0.000,B 14.930,C -40.070}
DECL LDAT LCPDATP183={VEL 1,ACC 100,APO_DIST 5,APO_FAC 50.0,ORI_TYP #VAR,CIRC_TYP #BASE,JERK_FAC 50.0}
DECL FDAT FP183={TOOL_NO 2,BASE_NO 10,IPO_FRAME #BASE,POINT2[] " ",TQ_STATE FALSE}
DECL E6POS XP183={X 59.570,Y 109.710,Z -37.080,A -0.000,B 18.740,C -38.660}
DECL LDAT LCPDATP184={VEL 1,ACC 100,APO_DIST 5,APO_FAC 50.0,ORI_TYP #VAR,CIRC_TYP #BASE,JERK_FAC 50.0}
DECL FDAT FP184={TOOL_NO 2,BASE_NO 10,IPO_FRAME #BASE,POINT2[] " ",TQ_STATE FALSE}
DECL E6POS XP184={X 60.010,Y 110.520,Z -38.420,A -0.000,B 17.860,C -36.410}
DECL LDAT LCPDATC185={VEL 0.1,ACC 100,APO_DIST 5,APO_FAC 50.0,ORI_TYP #VAR,CIRC_TYP #BASE,JERK_FAC 50.0}
DECL FDAT FC185={TOOL_NO 2,BASE_NO 10,IPO_FRAME #BASE,POINT2[] " ",TQ_STATE FALSE}
DECL E6POS XCAux185={X 48.130,Y 116.190,Z -38.420,A 0.000,B 14.240,C -37.780}
DECL E6POS XCDes185={X -48.130,Y 116.190,Z -38.420,A -0.000,B -14.240,C -37.780}
DECL LDAT LCPDATP186={VEL 1,ACC 100,APO_DIST 5,APO_FAC 50.0,ORI_TYP #VAR,CIRC_TYP #BASE,JERK_FAC 50.0}
DECL FDAT FP186={TOOL_NO 2,BASE_NO 10,IPO_FRAME #BASE,POINT2[] " ",TQ_STATE FALSE}
DECL E6POS XP186={X -60.010,Y 110.520,Z -38.420,A -0.000,B -17.860,C -36.410}
DECL LDAT LCPDATP187={VEL 1,ACC 100,APO_DIST 5,APO_FAC 50.0,ORI_TYP #VAR,CIRC_TYP #BASE,JERK_FAC 50.0}
DECL FDAT FP187={TOOL_NO 2,BASE_NO 10,IPO_FRAME #BASE,POINT2[] " ",TQ_STATE FALSE}
DECL E6POS XP187={X -62.870,Y 115.800,Z -42.570,A 0.000,B -13.520,C -26.280}
DECL LDAT LCPDATC188={VEL 0.1,ACC 100,APO_DIST 5,APO_FAC 50.0,ORI_TYP #VAR,CIRC_TYP #BASE,JERK_FAC 50.0}
DECL FDAT FC188={TOOL_NO 2,BASE_NO 10,IPO_FRAME #BASE,POINT2[] " ",TQ_STATE FALSE}
DECL E6POS XCAux188={X -50.430,Y 121.740,Z -42.570,A 0.000,B -10.810,C -27.440}
DECL E6POS XCDes188={X 50.430,Y 121.740,Z -42.570,A 0.000,B 10.810,C -27.440}
DECL LDAT LCPDATP189={VEL 1,ACC 100,APO_DIST 5,APO_FAC 50.0,ORI_TYP #VAR,CIRC_TYP #BASE,JERK_FAC 50.0}
DECL FDAT FP189={TOOL_NO 2,BASE_NO 10,IPO_FRAME #BASE,POINT2[] " ",TQ_STATE FALSE}
DECL E6POS XP189={X 62.870,Y 115.800,Z -42.570,A 0.000,B 13.520,C -26.280}
DECL LDAT LCPDATP190={VEL 1,ACC 100,APO_DIST 5,APO_FAC 50.0,ORI_TYP #VAR,CIRC_TYP #BASE,JERK_FAC 50.0}
DECL FDAT FP190={TOOL_NO 2,BASE_NO 10,IPO_FRAME #BASE,POINT2[] " ",TQ_STATE FALSE}
DECL E6POS XP190={X 66.060,Y 121.660,Z -45.540,A 0.000,B 8.780,C -16.530}
DECL LDAT LCPDATC191={VEL 0.1,ACC 100,APO_DIST 5,APO_FAC 50.0,ORI_TYP #VAR,CIRC_TYP #BASE,JERK_FAC 50.0}
DECL FDAT FC191={TOOL_NO 2,BASE_NO 10,IPO_FRAME #BASE,POINT2[] " ",TQ_STATE FALSE}
DECL E6POS XCAux191={X 52.980,Y 127.900,Z -45.540,A 0.000,B 7.030,C -17.330}
DECL E6POS XCDes191={X -52.980,Y 127.900,Z -45.540,A 0.000,B -7.030,C -17.330}
DECL LDAT LCPDATP192={VEL 1,ACC 100,APO_DIST 5,APO_FAC 50.0,ORI_TYP #VAR,CIRC_TYP #BASE,JERK_FAC 50.0}
DECL FDAT FP192={TOOL_NO 2,BASE_NO 10,IPO_FRAME #BASE,POINT2[] " ",TQ_STATE FALSE}
DECL E6POS XP192={X -66.060,Y 121.660,Z -45.540,A 0.000,B -8.780,C -16.530}
DECL LDAT LCPDATP193={VEL 1,ACC 100,APO_DIST 5,APO_FAC 50.0,ORI_TYP #VAR,CIRC_TYP #BASE,JERK_FAC 50.0}
DECL FDAT FP193={TOOL_NO 2,BASE_NO 10,IPO_FRAME #BASE,POINT2[] " ",TQ_STATE FALSE}
DECL E6POS XP193={X -69.440,Y 127.900,Z -47.220,A 0.000,B -3.810,C -7.040}
DECL LDAT LCPDATC194={VEL 0.1,ACC 100,APO_DIST 5,APO_FAC 50.0,ORI_TYP #VAR,CIRC_TYP #BASE,JERK_FAC 50.0}
DECL FDAT FC194={TOOL_NO 2,BASE_NO 10,IPO_FRAME #BASE,POINT2[] " ",TQ_STATE FALSE}
DECL E6POS XCAux194={X -55.690,Y 134.460,Z -47.220,A 0.000,B -3.050,C -7.400}
DECL E6POS XCDes194={X 55.690,Y 134.460,Z -47.220,A -0.000,B 3.050,C -7.400}
DECL LDAT LCPDATP195={VEL 1,ACC 100,APO_DIST 5,APO_FAC 50.0,ORI_TYP #VAR,CIRC_TYP #BASE,JERK_FAC 50.0}
DECL FDAT FP195={TOOL_NO 2,BASE_NO 10,IPO_FRAME #BASE,POINT2[] " ",TQ_STATE FALSE}
DECL E6POS XP195={X 69.440,Y 127.900,Z -47.220,A 0.000,B 3.810,C -7.040}
DECL LDAT LCPDATP196={VEL 1,ACC 100,APO_DIST 5,APO_FAC 50.0,ORI_TYP #VAR,CIRC_TYP #BASE,JERK_FAC 50.0}
DECL FDAT FP196={TOOL_NO 2,BASE_NO 10,IPO_FRAME #BASE,POINT2[] " ",TQ_STATE FALSE}
DECL E6POS XP196={X 71.810,Y 132.260,Z -47.600,A 0.000,B 0.000,C -0.000}
DECL LDAT LCPDATC197={VEL 0.1,ACC 100,APO_DIST 5,APO_FAC 50.0,ORI_TYP #VAR,CIRC_TYP #BASE,JERK_FAC 50.0}
DECL FDAT FC197={TOOL_NO 2,BASE_NO 10,IPO_FRAME #BASE,POINT2[] " ",TQ_STATE FALSE}
DECL E6POS XCAux197={X 57.590,Y 139.040,Z -47.600,A 0.000,B 0.000,C -0.000}
DECL E6POS XCDes197={X -57.590,Y 139.040,Z -47.600,A 0.000,B 0.000,C -0.000}
DECL LDAT LCPDATP198={VEL 1,ACC 100,APO_DIST 5,APO_FAC 50.0,ORI_TYP #VAR,CIRC_TYP #BASE,JERK_FAC 50.0}
DECL FDAT FP198={TOOL_NO 2,BASE_NO 10,IPO_FRAME #BASE,POINT2[] " ",TQ_STATE FALSE}
DECL E6POS XP198={X -71.810,Y 132.260,Z -47.600,A 0.000,B 0.000,C -0.000}
DECL LDAT LCPDATP199={VEL 1,ACC 100,APO_DIST 5,APO_FAC 50.0,ORI_TYP #VAR,CIRC_TYP #BASE,JERK_FAC 50.0}
DECL FDAT FP199={TOOL_NO 2,BASE_NO 10,IPO_FRAME #BASE,POINT2[] " ",TQ_STATE FALSE}
DECL E6POS XP199={X -70.860,Y 130.500,Z -47.600,A 0.000,B 0.000,C -0.000}
DECL LDAT LCPDATC200={VEL 0.1,ACC 100,APO_DIST 5,APO_FAC 50.0,ORI_TYP #VAR,CIRC_TYP #BASE,JERK_FAC 50.0}
DECL FDAT FC200={TOOL_NO 2,BASE_NO 10,IPO_FRAME #BASE,POINT2[] " ",TQ_STATE FALSE}
DECL E6POS XCAux200={X -56.830,Y 137.190,Z -47.600,A 0.000,B 0.000,C -0.000}
DECL E6POS XCDes200={X 56.830,Y 137.190,Z -47.600,A 0.000,B 0.000,C -0.000}
DECL LDAT LCPDATP201={VEL 1,ACC 100,APO_DIST 5,APO_FAC 50.0,ORI_TYP #VAR,CIRC_TYP #BASE,JERK_FAC 50.0}
DECL FDAT FP201={TOOL_NO 2,BASE_NO 10,IPO_FRAME #BASE,POINT2[] " ",TQ_STATE FALSE}
DECL E6POS XP201={X 70.860,Y 130.500,Z -47.600,A 0.000,B 0.000,C -0.000}
DECL LDAT LCPDATP202={VEL 1,ACC 100,APO_DIST 5,APO_FAC 50.0,ORI_TYP #VAR,CIRC_TYP #BASE,JERK_FAC 50.0}
DECL FDAT FP202={TOOL_NO 2,BASE_NO 10,IPO_FRAME #BASE,POINT2[] " ",TQ_STATE FALSE}
DECL E6POS XP202={X 69.900,Y 128.740,Z -47.600,A 0.000,B 0.000,C -0.000}
DECL LDAT LCPDATC203={VEL 0.1,ACC 100,APO_DIST 5,APO_FAC 50.0,ORI_TYP #VAR,CIRC_TYP #BASE,JERK_FAC 50.0}
DECL FDAT FC203={TOOL_NO 2,BASE_NO 10,IPO_FRAME #BASE,POINT2[] " ",TQ_STATE FALSE}
DECL E6POS XCAux203={X 56.060,Y 135.340,Z -47.600,A 0.000,B 0.000,C -0.000}
DECL E6POS XCDes203={X -56.060,Y 135.340,Z -47.600,A 0.000,B 0.000,C -0.000}
DECL LDAT LCPDATP204={VEL 1,ACC 100,APO_DIST 5,APO_FAC 50.0,ORI_TYP #VAR,CIRC_TYP #BASE,JERK_FAC 50.0}
DECL FDAT FP204={TOOL_NO 2,BASE_NO 10,IPO_FRAME #BASE,POINT2[] " ",TQ_STATE FALSE}
DECL E6POS XP204={X -69.900,Y 128.740,Z -47.600,A 0.000,B 0.000,C -0.000}
DECL LDAT LCPDATP205={VEL 1,ACC 100,APO_DIST 5,APO_FAC 50.0,ORI_TYP #VAR,CIRC_TYP #BASE,JERK_FAC 50.0}
DECL FDAT FP205={TOOL_NO 2,BASE_NO 10,IPO_FRAME #BASE,POINT2[] " ",TQ_STATE FALSE}
DECL E6POS XP205={X -68.950,Y 126.980,Z -47.600,A 0.000,B 0.000,C -0.000}
DECL LDAT LCPDATC206={VEL 0.1,ACC 100,APO_DIST 5,APO_FAC 50.0,ORI_TYP #VAR,CIRC_TYP #BASE,JERK_FAC 50.0}
DECL FDAT FC206={TOOL_NO 2,BASE_NO 10,IPO_FRAME #BASE,POINT2[] " ",TQ_STATE FALSE}
DECL E6POS XCAux206={X -55.300,Y 133.500,Z -47.600,A 0.000,B 0.000,C -0.000}
DECL E6POS XCDes206={X 55.300,Y 133.500,Z -47.600,A 0.000,B 0.000,C -0.000}
DECL LDAT LCPDATP207={VEL 1,ACC 100,APO_DIST 5,APO_FAC 50.0,ORI_TYP #VAR,CIRC_TYP #BASE,JERK_FAC 50.0}
DECL FDAT FP207={TOOL_NO 2,BASE_NO 10,IPO_FRAME #BASE,POINT2[] " ",TQ_STATE FALSE}
DECL E6POS XP207={X 68.950,Y 126.980,Z -47.600,A 0.000,B 0.000,C -0.000}
DECL LDAT LCPDATP208={VEL 1,ACC 100,APO_DIST 5,APO_FAC 50.0,ORI_TYP #VAR,CIRC_TYP #BASE,JERK_FAC 50.0}
DECL FDAT FP208={TOOL_NO 2,BASE_NO 10,IPO_FRAME #BASE,POINT2[] " ",TQ_STATE FALSE}
DECL E6POS XP208={X 67.990,Y 125.230,Z -47.600,A 0.000,B 0.000,C -0.000}
DECL LDAT LCPDATC209={VEL 0.1,ACC 100,APO_DIST 5,APO_FAC 50.0,ORI_TYP #VAR,CIRC_TYP #BASE,JERK_FAC 50.0}
DECL FDAT FC209={TOOL_NO 2,BASE_NO 10,IPO_FRAME #BASE,POINT2[] " ",TQ_STATE FALSE}
DECL E6POS XCAux209={X 54.530,Y 131.650,Z -47.600,A 0.000,B 0.000,C -0.000}
DECL E6POS XCDes209={X -54.530,Y 131.650,Z -47.600,A 0.000,B 0.000,C -0.000}
DECL LDAT LCPDATP210={VEL 1,ACC 100,APO_DIST 5,APO_FAC 50.0,ORI_TYP #VAR,CIRC_TYP #BASE,JERK_FAC 50.0}
DECL FDAT FP210={TOOL_NO 2,BASE_NO 10,IPO_FRAME #BASE,POINT2[] " ",TQ_STATE FALSE}
DECL E6POS XP210={X -67.990,Y 125.230,Z -47.600,A 0.000,B 0.000,C -0.000}
DECL LDAT LCPDATP211={VEL 1,ACC 100,APO_DIST 5,APO_FAC 50.0,ORI_TYP #VAR,CIRC_TYP #BASE,JERK_FAC 50.0}
DECL FDAT FP211={TOOL_NO 2,BASE_NO 10,IPO_FRAME #BASE,POINT2[] " ",TQ_STATE FALSE}
DECL E6POS XP211={X -67.040,Y 123.470,Z -47.600,A 0.000,B 0.000,C -0.000}
DECL LDAT LCPDATC212={VEL 0.1,ACC 100,APO_DIST 5,APO_FAC 50.0,ORI_TYP #VAR,CIRC_TYP #BASE,JERK_FAC 50.0}
DECL FDAT FC212={TOOL_NO 2,BASE_NO 10,IPO_FRAME #BASE,POINT2[] " ",TQ_STATE FALSE}
DECL E6POS XCAux212={X -53.760,Y 129.800,Z -47.600,A 0.000,B 0.000,C -0.000}
DECL E6POS XCDes212={X 53.760,Y 129.800,Z -47.600,A 0.000,B 0.000,C -0.000}
DECL LDAT LCPDATP213={VEL 1,ACC 100,APO_DIST 5,APO_FAC 50.0,ORI_TYP #VAR,CIRC_TYP #BASE,JERK_FAC 50.0}
DECL FDAT FP213={TOOL_NO 2,BASE_NO 10,IPO_FRAME #BASE,POINT2[] " ",TQ_STATE FALSE}
DECL E6POS XP213={X 67.040,Y 123.470,Z -47.600,A 0.000,B 0.000,C -0.000}
DECL LDAT LCPDATP214={VEL 1,ACC 100,APO_DIST 5,APO_FAC 50.0,ORI_TYP #VAR,CIRC_TYP #BASE,JERK_FAC 50.0}
DECL FDAT FP214={TOOL_NO 2,BASE_NO 10,IPO_FRAME #BASE,POINT2[] " ",TQ_STATE FALSE}
DECL E6POS XP214={X 67.210,Y 123.780,Z -47.560,A 0.000,B -1.290,C 2.370}
DECL LDAT LCPDATC215={VEL 0.1,ACC 100,APO_DIST 5,APO_FAC 50.0,ORI_TYP #VAR,CIRC_TYP #BASE,JERK_FAC 50.0}
DECL FDAT FC215={TOOL_NO 2,BASE_NO 10,IPO_FRAME #BASE,POINT2[] " ",TQ_STATE FALSE}
DECL E6POS XCAux215={X 53.900,Y 130.130,Z -47.560,A 0.000,B -1.030,C 2.490}
DECL E6POS XCDes215={X -53.900,Y 130.130,Z -47.560,A 0.000,B 1.030,C 2.490}
DECL LDAT LCPDATP216={VEL 1,ACC 100,APO_DIST 5,APO_FAC 50.0,ORI_TYP #VAR,CIRC_TYP #BASE,JERK_FAC 50.0}
DECL FDAT FP216={TOOL_NO 2,BASE_NO 10,IPO_FRAME #BASE,POINT2[] " ",TQ_STATE FALSE}
DECL E6POS XP216={X -67.210,Y 123.780,Z -47.560,A -0.000,B 1.290,C 2.370}
DECL LDAT LCPDATP217={VEL 1,ACC 100,APO_DIST 5,APO_FAC 50.0,ORI_TYP #VAR,CIRC_TYP #BASE,JERK_FAC 50.0}
DECL FDAT FP217={TOOL_NO 2,BASE_NO 10,IPO_FRAME #BASE,POINT2[] " ",TQ_STATE FALSE}
DECL E6POS XP217={X -70.650,Y 130.130,Z -46.540,A -0.000,B 6.330,C 11.790}
DECL LDAT LCPDATC218={VEL 0.1,ACC 100,APO_DIST 5,APO_FAC 50.0,ORI_TYP #VAR,CIRC_TYP #BASE,JERK_FAC 50.0}
DECL FDAT FC218={TOOL_NO 2,BASE_NO 10,IPO_FRAME #BASE,POINT2[] " ",TQ_STATE FALSE}
DECL E6POS XCAux218={X -56.670,Y 136.800,Z -46.540,A -0.000,B 5.070,C 12.380}
DECL E6POS XCDes218={X 56.670,Y 136.800,Z -46.540,A -0.000,B -5.070,C 12.380}
DECL LDAT LCPDATP219={VEL 1,ACC 100,APO_DIST 5,APO_FAC 50.0,ORI_TYP #VAR,CIRC_TYP #BASE,JERK_FAC 50.0}
DECL FDAT FP219={TOOL_NO 2,BASE_NO 10,IPO_FRAME #BASE,POINT2[] " ",TQ_STATE FALSE}
DECL E6POS XP219={X 70.650,Y 130.130,Z -46.540,A 0.000,B -6.330,C 11.790}
DECL LDAT LCPDATP220={VEL 1,ACC 100,APO_DIST 5,APO_FAC 50.0,ORI_TYP #VAR,CIRC_TYP #BASE,JERK_FAC 50.0}
DECL FDAT FP220={TOOL_NO 2,BASE_NO 10,IPO_FRAME #BASE,POINT2[] " ",TQ_STATE FALSE}
DECL E6POS XP220={X 73.950,Y 136.210,Z -44.200,A 0.000,B -11.200,C 21.400}
DECL LDAT LCPDATC221={VEL 0.1,ACC 100,APO_DIST 5,APO_FAC 50.0,ORI_TYP #VAR,CIRC_TYP #BASE,JERK_FAC 50.0}
DECL FDAT FC221={TOOL_NO 2,BASE_NO 10,IPO_FRAME #BASE,POINT2[] " ",TQ_STATE FALSE}
DECL E6POS XCAux221={X 59.310,Y 143.190,Z -44.200,A -0.000,B -8.970,C 22.390}
DECL E6POS XCDes221={X -59.310,Y 143.190,Z -44.200,A 0.000,B 8.970,C 22.390}
DECL LDAT LCPDATP222={VEL 1,ACC 100,APO_DIST 5,APO_FAC 50.0,ORI_TYP #VAR,CIRC_TYP #BASE,JERK_FAC 50.0}
DECL FDAT FP222={TOOL_NO 2,BASE_NO 10,IPO_FRAME #BASE,POINT2[] " ",TQ_STATE FALSE}
DECL E6POS XP222={X -73.950,Y 136.210,Z -44.200,A 0.000,B 11.200,C 21.400}
DECL LDAT LCPDATP223={VEL 1,ACC 100,APO_DIST 5,APO_FAC 50.0,ORI_TYP #VAR,CIRC_TYP #BASE,JERK_FAC 50.0}
DECL FDAT FP223={TOOL_NO 2,BASE_NO 10,IPO_FRAME #BASE,POINT2[] " ",TQ_STATE FALSE}
DECL E6POS XP223={X -76.990,Y 141.800,Z -40.620,A 0.000,B 15.760,C 31.320}
DECL LDAT LCPDATC224={VEL 0.1,ACC 100,APO_DIST 5,APO_FAC 50.0,ORI_TYP #VAR,CIRC_TYP #BASE,JERK_FAC 50.0}
DECL FDAT FC224={TOOL_NO 2,BASE_NO 10,IPO_FRAME #BASE,POINT2[] " ",TQ_STATE FALSE}
DECL E6POS XCAux224={X -61.750,Y 149.070,Z -40.620,A 0.000,B 12.580,C 32.610}
DECL E6POS XCDes224={X 61.750,Y 149.070,Z -40.620,A 0.000,B -12.580,C 32.610}
DECL LDAT LCPDATP225={VEL 1,ACC 100,APO_DIST 5,APO_FAC 50.0,ORI_TYP #VAR,CIRC_TYP #BASE,JERK_FAC 50.0}
DECL FDAT FP225={TOOL_NO 2,BASE_NO 10,IPO_FRAME #BASE,POINT2[] " ",TQ_STATE FALSE}
DECL E6POS XP225={X 76.990,Y 141.800,Z -40.620,A 0.000,B -15.760,C 31.320}
DECL LDAT LCPDATP226={VEL 1,ACC 100,APO_DIST 5,APO_FAC 50.0,ORI_TYP #VAR,CIRC_TYP #BASE,JERK_FAC 50.0}
DECL FDAT FP226={TOOL_NO 2,BASE_NO 10,IPO_FRAME #BASE,POINT2[] " ",TQ_STATE FALSE}
DECL E6POS XP226={X 79.650,Y 146.710,Z -35.920,A 0.000,B -19.850,C 41.670}
DECL LDAT LCPDATC227={VEL 0.1,ACC 100,APO_DIST 5,APO_FAC 50.0,ORI_TYP #VAR,CIRC_TYP #BASE,JERK_FAC 50.0}
DECL FDAT FC227={TOOL_NO 2,BASE_NO 10,IPO_FRAME #BASE,POINT2[] " ",TQ_STATE FALSE}
DECL E6POS XCAux227={X 63.880,Y 154.230,Z -35.920,A 0.000,B -15.800,C 43.100}
DECL E6POS XCDes227={X -63.880,Y 154.230,Z -35.920,A 0.000,B 15.800,C 43.100}
DECL LDAT LCPDATP228={VEL 1,ACC 100,APO_DIST 5,APO_FAC 50.0,ORI_TYP #VAR,CIRC_TYP #BASE,JERK_FAC 50.0}
DECL FDAT FP228={TOOL_NO 2,BASE_NO 10,IPO_FRAME #BASE,POINT2[] " ",TQ_STATE FALSE}
DECL E6POS XP228={X -79.650,Y 146.710,Z -35.920,A 0.000,B 19.850,C 41.670}
DECL LDAT LCPDATP229={VEL 1,ACC 100,APO_DIST 5,APO_FAC 50.0,ORI_TYP #VAR,CIRC_TYP #BASE,JERK_FAC 50.0}
DECL FDAT FP229={TOOL_NO 2,BASE_NO 10,IPO_FRAME #BASE,POINT2[] " ",TQ_STATE FALSE}
DECL E6POS XP229={X -78.490,Y 144.560,Z -38.720,A -0.000,B 17.860,C 36.410}
DECL LDAT LCPDATC230={VEL 0.1,ACC 100,APO_DIST 5,APO_FAC 50.0,ORI_TYP #VAR,CIRC_TYP #BASE,JERK_FAC 50.0}
DECL FDAT FC230={TOOL_NO 2,BASE_NO 10,IPO_FRAME #BASE,POINT2[] " ",TQ_STATE FALSE}
DECL E6POS XCAux230={X -62.950,Y 151.970,Z -38.720,A -0.000,B 14.240,C 37.780}
DECL E6POS XCDes230={X 62.950,Y 151.970,Z -38.720,A 0.000,B -14.240,C 37.780}
DECL LDAT LCPDATP231={VEL 1,ACC 100,APO_DIST 5,APO_FAC 50.0,ORI_TYP #VAR,CIRC_TYP #BASE,JERK_FAC 50.0}
DECL FDAT FP231={TOOL_NO 2,BASE_NO 10,IPO_FRAME #BASE,POINT2[] " ",TQ_STATE FALSE}
DECL E6POS XP231={X 78.490,Y 144.560,Z -38.720,A -0.000,B -17.860,C 36.410}
DECL LDAT LCPDATP232={VEL 1,ACC 100,APO_DIST 5,APO_FAC 50.0,ORI_TYP #VAR,CIRC_TYP #BASE,JERK_FAC 50.0}
DECL FDAT FP232={TOOL_NO 2,BASE_NO 10,IPO_FRAME #BASE,POINT2[] " ",TQ_STATE FALSE}
DECL E6POS XP232={X 75.480,Y 139.010,Z -43.050,A -0.000,B -13.340,C 25.900}
DECL LDAT LCPDATC233={VEL 0.1,ACC 100,APO_DIST 5,APO_FAC 50.0,ORI_TYP #VAR,CIRC_TYP #BASE,JERK_FAC 50.0}
DECL FDAT FC233={TOOL_NO 2,BASE_NO 10,IPO_FRAME #BASE,POINT2[] " ",TQ_STATE FALSE}
DECL E6POS XCAux233={X 60.530,Y 146.140,Z -43.050,A 0.000,B -10.660,C 27.040}
DECL E6POS XCDes233={X -60.530,Y 146.140,Z -43.050,A 0.000,B 10.660,C 27.040}
DECL LDAT LCPDATP234={VEL 1,ACC 100,APO_DIST 5,APO_FAC 50.0,ORI_TYP #VAR,CIRC_TYP #BASE,JERK_FAC 50.0}
DECL FDAT FP234={TOOL_NO 2,BASE_NO 10,IPO_FRAME #BASE,POINT2[] " ",TQ_STATE FALSE}
DECL E6POS XP234={X -75.480,Y 139.010,Z -43.050,A -0.000,B 13.340,C 25.900}
DECL LDAT LCPDATP235={VEL 1,ACC 100,APO_DIST 5,APO_FAC 50.0,ORI_TYP #VAR,CIRC_TYP #BASE,JERK_FAC 50.0}
DECL FDAT FP235={TOOL_NO 2,BASE_NO 10,IPO_FRAME #BASE,POINT2[] " ",TQ_STATE FALSE}
DECL E6POS XP235={X -72.120,Y 132.830,Z -46.090,A 0.000,B 8.410,C 15.790}
DECL LDAT LCPDATC236={VEL 0.1,ACC 100,APO_DIST 5,APO_FAC 50.0,ORI_TYP #VAR,CIRC_TYP #BASE,JERK_FAC 50.0}
DECL FDAT FC236={TOOL_NO 2,BASE_NO 10,IPO_FRAME #BASE,POINT2[] " ",TQ_STATE FALSE}
DECL E6POS XCAux236={X -57.840,Y 139.640,Z -46.090,A 0.000,B 6.730,C 16.560}
DECL E6POS XCDes236={X 57.840,Y 139.640,Z -46.090,A 0.000,B -6.730,C 16.560}
DECL LDAT LCPDATP237={VEL 1,ACC 100,APO_DIST 5,APO_FAC 50.0,ORI_TYP #VAR,CIRC_TYP #BASE,JERK_FAC 50.0}
DECL FDAT FP237={TOOL_NO 2,BASE_NO 10,IPO_FRAME #BASE,POINT2[] " ",TQ_STATE FALSE}
DECL E6POS XP237={X 72.120,Y 132.830,Z -46.090,A 0.000,B -8.410,C 15.790}
DECL LDAT LCPDATP238={VEL 1,ACC 100,APO_DIST 5,APO_FAC 50.0,ORI_TYP #VAR,CIRC_TYP #BASE,JERK_FAC 50.0}
DECL FDAT FP238={TOOL_NO 2,BASE_NO 10,IPO_FRAME #BASE,POINT2[] " ",TQ_STATE FALSE}
DECL E6POS XP238={X 68.550,Y 126.260,Z -47.720,A 0.000,B -3.220,C 5.950}
DECL LDAT LCPDATC239={VEL 0.1,ACC 100,APO_DIST 5,APO_FAC 50.0,ORI_TYP #VAR,CIRC_TYP #BASE,JERK_FAC 50.0}
DECL FDAT FC239={TOOL_NO 2,BASE_NO 10,IPO_FRAME #BASE,POINT2[] " ",TQ_STATE FALSE}
DECL E6POS XCAux239={X 54.980,Y 132.730,Z -47.720,A 0.000,B -2.580,C 6.250}
DECL E6POS XCDes239={X -54.980,Y 132.730,Z -47.720,A 0.000,B 2.580,C 6.250}
DECL LDAT LCPDATP240={VEL 1,ACC 100,APO_DIST 5,APO_FAC 50.0,ORI_TYP #VAR,CIRC_TYP #BASE,JERK_FAC 50.0}
DECL FDAT FP240={TOOL_NO 2,BASE_NO 10,IPO_FRAME #BASE,POINT2[] " ",TQ_STATE FALSE}
DECL E6POS XP240={X -68.550,Y 126.260,Z -47.720,A 0.000,B 3.220,C 5.950}
DECL LDAT LCPDATP241={VEL 1,ACC 100,APO_DIST 5,APO_FAC 50.0,ORI_TYP #VAR,CIRC_TYP #BASE,JERK_FAC 50.0}
DECL FDAT FP241={TOOL_NO 2,BASE_NO 10,IPO_FRAME #BASE,POINT2[] " ",TQ_STATE FALSE}
DECL E6POS XP241={X -66.700,Y 122.840,Z -48.000,A 0.000,B 0.000,C -0.000}
DECL LDAT LCPDATC242={VEL 0.1,ACC 100,APO_DIST 5,APO_FAC 50.0,ORI_TYP #VAR,CIRC_TYP #BASE,JERK_FAC 50.0}
DECL FDAT FC242={TOOL_NO 2,BASE_NO 10,IPO_FRAME #BASE,POINT2[] " ",TQ_STATE FALSE}
DECL E6POS XCAux242={X -53.490,Y 129.140,Z -48.000,A 0.000,B 0.000,C -0.000}
DECL E6POS XCDes242={X 53.490,Y 129.140,Z -48.000,A 0.000,B 0.000,C -0.000}
DECL LDAT LCPDATP243={VEL 1,ACC 100,APO_DIST 5,APO_FAC 50.0,ORI_TYP #VAR,CIRC_TYP #BASE,JERK_FAC 50.0}
DECL FDAT FP243={TOOL_NO 2,BASE_NO 10,IPO_FRAME #BASE,POINT2[] " ",TQ_STATE FALSE}
DECL E6POS XP243={X 66.700,Y 122.840,Z -48.000,A 0.000,B 0.000,C -0.000}
DECL LDAT LCPDATP244={VEL 1,ACC 100,APO_DIST 5,APO_FAC 50.0,ORI_TYP #VAR,CIRC_TYP #BASE,JERK_FAC 50.0}
DECL FDAT FP244={TOOL_NO 2,BASE_NO 10,IPO_FRAME #BASE,POINT2[] " ",TQ_STATE FALSE}
DECL E6POS XP244={X 67.650,Y 124.600,Z -48.000,A 0.000,B 0.000,C -0.000}
DECL LDAT LCPDATC245={VEL 0.1,ACC 100,APO_DIST 5,APO_FAC 50.0,ORI_TYP #VAR,CIRC_TYP #BASE,JERK_FAC 50.0}
DECL FDAT FC245={TOOL_NO 2,BASE_NO 10,IPO_FRAME #BASE,POINT2[] " ",TQ_STATE FALSE}
DECL E6POS XCAux245={X 54.260,Y 130.990,Z -48.000,A 0.000,B 0.000,C -0.000}
DECL E6POS XCDes245={X -54.260,Y 130.990,Z -48.000,A 0.000,B 0.000,C -0.000}
DECL LDAT LCPDATP246={VEL 1,ACC 100,APO_DIST 5,APO_FAC 50.0,ORI_TYP #VAR,CIRC_TYP #BASE,JERK_FAC 50.0}
DECL FDAT FP246={TOOL_NO 2,BASE_NO 10,IPO_FRAME #BASE,POINT2[] " ",TQ_STATE FALSE}
DECL E6POS XP246={X -67.650,Y 124.600,Z -48.000,A 0.000,B 0.000,C -0.000}
DECL LDAT LCPDATP247={VEL 1,ACC 100,APO_DIST 5,APO_FAC 50.0,ORI_TYP #VAR,CIRC_TYP #BASE,JERK_FAC 50.0}
DECL FDAT FP247={TOOL_NO 2,BASE_NO 10,IPO_FRAME #BASE,POINT2[] " ",TQ_STATE FALSE}
DECL E6POS XP247={X -68.610,Y 126.360,Z -48.000,A 0.000,B 0.000,C -0.000}
DECL LDAT LCPDATC248={VEL 0.1,ACC 100,APO_DIST 5,APO_FAC 50.0,ORI_TYP #VAR,CIRC_TYP #BASE,JERK_FAC 50.0}
DECL FDAT FC248={TOOL_NO 2,BASE_NO 10,IPO_FRAME #BASE,POINT2[] " ",TQ_STATE FALSE}
DECL E6POS XCAux248={X -55.020,Y 132.840,Z -48.000,A 0.000,B 0.000,C -0.000}
DECL E6POS XCDes248={X 55.020,Y 132.840,Z -48.000,A 0.000,B 0.000,C -0.000}
DECL LDAT LCPDATP249={VEL 1,ACC 100,APO_DIST 5,APO_FAC 50.0,ORI_TYP #VAR,CIRC_TYP #BASE,JERK_FAC 50.0}
DECL FDAT FP249={TOOL_NO 2,BASE_NO 10,IPO_FRAME #BASE,POINT2[] " ",TQ_STATE FALSE}
DECL E6POS XP249={X 68.610,Y 126.360,Z -48.000,A 0.000,B 0.000,C -0.000}
DECL LDAT LCPDATP250={VEL 1,ACC 100,APO_DIST 5,APO_FAC 50.0,ORI_TYP #VAR,CIRC_TYP #BASE,JERK_FAC 50.0}
DECL FDAT FP250={TOOL_NO 2,BASE_NO 10,IPO_FRAME #BASE,POINT2[] " ",TQ_STATE FALSE}
DECL E6POS XP250={X 69.560,Y 128.120,Z -48.000,A 0.000,B 0.000,C -0.000}
DECL LDAT LCPDATC251={VEL 0.1,ACC 100,APO_DIST 5,APO_FAC 50.0,ORI_TYP #VAR,CIRC_TYP #BASE,JERK_FAC 50.0}
DECL FDAT FC251={TOOL_NO 2,BASE_NO 10,IPO_FRAME #BASE,POINT2[] " ",TQ_STATE FALSE}
DECL E6POS XCAux251={X 55.790,Y 134.690,Z -48.000,A 0.000,B 0.000,C -0.000}
DECL E6POS XCDes251={X -55.790,Y 134.690,Z -48.000,A 0.000,B 0.000,C -0.000}
DECL LDAT LCPDATP252={VEL 1,ACC 100,APO_DIST 5,APO_FAC 50.0,ORI_TYP #VAR,CIRC_TYP #BASE,JERK_FAC 50.0}
DECL FDAT FP252={TOOL_NO 2,BASE_NO 10,IPO_FRAME #BASE,POINT2[] " ",TQ_STATE FALSE}
DECL E6POS XP252={X -69.560,Y 128.120,Z -48.000,A 0.000,B 0.000,C -0.000}
DECL LDAT LCPDATP253={VEL 1,ACC 100,APO_DIST 5,APO_FAC 50.0,ORI_TYP #VAR,CIRC_TYP #BASE,JERK_FAC 50.0}
DECL FDAT FP253={TOOL_NO 2,BASE_NO 10,IPO_FRAME #BASE,POINT2[] " ",TQ_STATE FALSE}
DECL E6POS XP253={X -70.520,Y 129.870,Z -48.000,A 0.000,B 0.000,C -0.000}
DECL LDAT LCPDATC254={VEL 0.1,ACC 100,APO_DIST 5,APO_FAC 50.0,ORI_TYP #VAR,CIRC_TYP #BASE,JERK_FAC 50.0}
DECL FDAT FC254={TOOL_NO 2,BASE_NO 10,IPO_FRAME #BASE,POINT2[] " ",TQ_STATE FALSE}
DECL E6POS XCAux254={X -56.550,Y 136.530,Z -48.000,A 0.000,B 0.000,C -0.000}
DECL E6POS XCDes254={X 56.550,Y 136.530,Z -48.000,A 0.000,B 0.000,C -0.000}
DECL LDAT LCPDATP255={VEL 1,ACC 100,APO_DIST 5,APO_FAC 50.0,ORI_TYP #VAR,CIRC_TYP #BASE,JERK_FAC 50.0}
DECL FDAT FP255={TOOL_NO 2,BASE_NO 10,IPO_FRAME #BASE,POINT2[] " ",TQ_STATE FALSE}
DECL E6POS XP255={X 70.520,Y 129.870,Z -48.000,A 0.000,B 0.000,C -0.000}
DECL LDAT LCPDATP256={VEL 1,ACC 100,APO_DIST 5,APO_FAC 50.0,ORI_TYP #VAR,CIRC_TYP #BASE,JERK_FAC 50.0}
DECL FDAT FP256={TOOL_NO 2,BASE_NO 10,IPO_FRAME #BASE,POINT2[] " ",TQ_STATE FALSE}
DECL E6POS XP256={X 71.470,Y 131.630,Z -48.000,A 0.000,B 0.000,C -0.000}
DECL LDAT LCPDATC257={VEL 0.1,ACC 100,APO_DIST 5,APO_FAC 50.0,ORI_TYP #VAR,CIRC_TYP #BASE,JERK_FAC 50.0}
DECL FDAT FC257={TOOL_NO 2,BASE_NO 10,IPO_FRAME #BASE,POINT2[] " ",TQ_STATE FALSE}
DECL E6POS XCAux257={X 57.320,Y 138.380,Z -48.000,A 0.000,B 0.000,C -0.000}
DECL E6POS XCDes257={X -57.320,Y 138.380,Z -48.000,A 0.000,B 0.000,C -0.000}
DECL LDAT LCPDATP258={VEL 1,ACC 100,APO_DIST 5,APO_FAC 50.0,ORI_TYP #VAR,CIRC_TYP #BASE,JERK_FAC 50.0}
DECL FDAT FP258={TOOL_NO 2,BASE_NO 10,IPO_FRAME #BASE,POINT2[] " ",TQ_STATE FALSE}
DECL E6POS XP258={X -71.470,Y 131.630,Z -48.000,A 0.000,B 0.000,C -0.000}
DECL LDAT LCPDATP259={VEL 1,ACC 100,APO_DIST 5,APO_FAC 50.0,ORI_TYP #VAR,CIRC_TYP #BASE,JERK_FAC 50.0}
DECL FDAT FP259={TOOL_NO 2,BASE_NO 10,IPO_FRAME #BASE,POINT2[] " ",TQ_STATE FALSE}
DECL E6POS XP259={X -70.620,Y 130.060,Z -47.890,A 0.000,B -2.070,C -3.820}
DECL LDAT LCPDATC260={VEL 0.1,ACC 100,APO_DIST 5,APO_FAC 50.0,ORI_TYP #VAR,CIRC_TYP #BASE,JERK_FAC 50.0}
DECL FDAT FC260={TOOL_NO 2,BASE_NO 10,IPO_FRAME #BASE,POINT2[] " ",TQ_STATE FALSE}
DECL E6POS XCAux260={X -56.640,Y 136.730,Z -47.890,A 0.000,B -1.660,C -4.010}
DECL E6POS XCDes260={X 56.640,Y 136.730,Z -47.890,A -0.000,B 1.660,C -4.010}
DECL LDAT LCPDATP261={VEL 1,ACC 100,APO_DIST 5,APO_FAC 50.0,ORI_TYP #VAR,CIRC_TYP #BASE,JERK_FAC 50.0}
DECL FDAT FP261={TOOL_NO 2,BASE_NO 10,IPO_FRAME #BASE,POINT2[] " ",TQ_STATE FALSE}
DECL E6POS XP261={X 70.620,Y 130.060,Z -47.890,A 0.000,B 2.070,C -3.820}
DECL LDAT LCPDATP262={VEL 1,ACC 100,APO_DIST 5,APO_FAC 50.0,ORI_TYP #VAR,CIRC_TYP #BASE,JERK_FAC 50.0}
DECL FDAT FP262={TOOL_NO 2,BASE_NO 10,IPO_FRAME #BASE,POINT2[] " ",TQ_STATE FALSE}
DECL E6POS XP262={X 67.020,Y 123.430,Z -46.570,A -0.000,B 7.290,C -13.620}
DECL LDAT LCPDATC263={VEL 0.1,ACC 100,APO_DIST 5,APO_FAC 50.0,ORI_TYP #VAR,CIRC_TYP #BASE,JERK_FAC 50.0}
DECL FDAT FC263={TOOL_NO 2,BASE_NO 10,IPO_FRAME #BASE,POINT2[] " ",TQ_STATE FALSE}
DECL E6POS XCAux263={X 53.750,Y 129.760,Z -46.570,A 0.000,B 5.840,C -14.300}
DECL E6POS XCDes263={X -53.750,Y 129.760,Z -46.570,A -0.000,B -5.840,C -14.300}
DECL LDAT LCPDATP264={VEL 1,ACC 100,APO_DIST 5,APO_FAC 50.0,ORI_TYP #VAR,CIRC_TYP #BASE,JERK_FAC 50.0}
DECL FDAT FP264={TOOL_NO 2,BASE_NO 10,IPO_FRAME #BASE,POINT2[] " ",TQ_STATE FALSE}
DECL E6POS XP264={X -67.020,Y 123.430,Z -46.570,A 0.000,B -7.290,C -13.620}
DECL LDAT LCPDATP265={VEL 1,ACC 100,APO_DIST 5,APO_FAC 50.0,ORI_TYP #VAR,CIRC_TYP #BASE,JERK_FAC 50.0}
DECL FDAT FP265={TOOL_NO 2,BASE_NO 10,IPO_FRAME #BASE,POINT2[] " ",TQ_STATE FALSE}
DECL E6POS XP265={X -63.610,Y 117.150,Z -43.830,A 0.000,B -12.290,C -23.660}
DECL LDAT LCPDATC266={VEL 0.1,ACC 100,APO_DIST 5,APO_FAC 50.0,ORI_TYP #VAR,CIRC_TYP #BASE,JERK_FAC 50.0}
DECL FDAT FC266={TOOL_NO 2,BASE_NO 10,IPO_FRAME #BASE,POINT2[] " ",TQ_STATE FALSE}
DECL E6POS XCAux266={X -51.010,Y 123.160,Z -43.830,A -0.000,B -9.830,C -24.730}
DECL E6POS XCDes266={X 51.010,Y 123.160,Z -43.830,A 0.000,B 9.830,C -24.730}
DECL LDAT LCPDATP267={VEL 1,ACC 100,APO_DIST 5,APO_FAC 50.0,ORI_TYP #VAR,CIRC_TYP #BASE,JERK_FAC 50.0}
DECL FDAT FP267={TOOL_NO 2,BASE_NO 10,IPO_FRAME #BASE,POINT2[] " ",TQ_STATE FALSE}
DECL E6POS XP267={X 63.610,Y 117.150,Z -43.830,A 0.000,B 12.290,C -23.660}
DECL LDAT LCPDATP268={VEL 1,ACC 100,APO_DIST 5,APO_FAC 50.0,ORI_TYP #VAR,CIRC_TYP #BASE,JERK_FAC 50.0}
DECL FDAT FP268={TOOL_NO 2,BASE_NO 10,IPO_FRAME #BASE,POINT2[] " ",TQ_STATE FALSE}
DECL E6POS XP268={X 60.510,Y 111.450,Z -39.770,A 0.000,B 16.920,C -34.070}
DECL LDAT LCPDATC269={VEL 0.1,ACC 100,APO_DIST 5,APO_FAC 50.0,ORI_TYP #VAR,CIRC_TYP #BASE,JERK_FAC 50.0}
DECL FDAT FC269={TOOL_NO 2,BASE_NO 10,IPO_FRAME #BASE,POINT2[] " ",TQ_STATE FALSE}
DECL E6POS XCAux269={X 48.530,Y 117.160,Z -39.770,A 0.000,B 13.500,C -35.410}
DECL E6POS XCDes269={X -48.530,Y 117.160,Z -39.770,A 0.000,B -13.500,C -35.410}
DECL LDAT LCPDATP270={VEL 1,ACC 100,APO_DIST 5,APO_FAC 50.0,ORI_TYP #VAR,CIRC_TYP #BASE,JERK_FAC 50.0}
DECL FDAT FP270={TOOL_NO 2,BASE_NO 10,IPO_FRAME #BASE,POINT2[] " ",TQ_STATE FALSE}
DECL E6POS XP270={X -60.510,Y 111.450,Z -39.770,A 0.000,B -16.920,C -34.070}
DECL LDAT LCPDATP271={VEL 1,ACC 100,APO_DIST 5,APO_FAC 50.0,ORI_TYP #VAR,CIRC_TYP #BASE,JERK_FAC 50.0}
DECL FDAT FP271={TOOL_NO 2,BASE_NO 10,IPO_FRAME #BASE,POINT2[] " ",TQ_STATE FALSE}
DECL E6POS XP271={X -59.760,Y 110.070,Z -39.030,A 0.000,B -17.860,C -36.410}
DECL LDAT LCPDATC272={VEL 0.1,ACC 100,APO_DIST 5,APO_FAC 50.0,ORI_TYP #VAR,CIRC_TYP #BASE,JERK_FAC 50.0}
DECL FDAT FC272={TOOL_NO 2,BASE_NO 10,IPO_FRAME #BASE,POINT2[] " ",TQ_STATE FALSE}
DECL E6POS XCAux272={X -47.930,Y 115.720,Z -39.030,A 0.000,B -14.240,C -37.780}
DECL E6POS XCDes272={X 47.930,Y 115.720,Z -39.030,A 0.000,B 14.240,C -37.780}
DECL LDAT LCPDATP273={VEL 1,ACC 100,APO_DIST 5,APO_FAC 50.0,ORI_TYP #VAR,CIRC_TYP #BASE,JERK_FAC 50.0}
DECL FDAT FP273={TOOL_NO 2,BASE_NO 10,IPO_FRAME #BASE,POINT2[] " ",TQ_STATE FALSE}
DECL E6POS XP273={X 59.760,Y 110.070,Z -39.030,A 0.000,B 17.860,C -36.410}
DECL LDAT LCPDATP274={VEL 1,ACC 100,APO_DIST 5,APO_FAC 50.0,ORI_TYP #VAR,CIRC_TYP #BASE,JERK_FAC 50.0}
DECL FDAT FP274={TOOL_NO 2,BASE_NO 10,IPO_FRAME #BASE,POINT2[] " ",TQ_STATE FALSE}
DECL E6POS XP274={X 62.940,Y 115.920,Z -43.550,A 0.000,B 13.150,C -25.480}
DECL LDAT LCPDATC275={VEL 0.1,ACC 100,APO_DIST 5,APO_FAC 50.0,ORI_TYP #VAR,CIRC_TYP #BASE,JERK_FAC 50.0}
DECL FDAT FC275={TOOL_NO 2,BASE_NO 10,IPO_FRAME #BASE,POINT2[] " ",TQ_STATE FALSE}
DECL E6POS XCAux275={X 50.480,Y 121.860,Z -43.550,A 0.000,B 10.510,C -26.610}
DECL E6POS XCDes275={X -50.480,Y 121.860,Z -43.550,A 0.000,B -10.510,C -26.610}
DECL LDAT LCPDATP276={VEL 1,ACC 100,APO_DIST 5,APO_FAC 50.0,ORI_TYP #VAR,CIRC_TYP #BASE,JERK_FAC 50.0}
DECL FDAT FP276={TOOL_NO 2,BASE_NO 10,IPO_FRAME #BASE,POINT2[] " ",TQ_STATE FALSE}
DECL E6POS XP276={X -62.940,Y 115.920,Z -43.550,A 0.000,B -13.150,C -25.480}
DECL LDAT LCPDATP277={VEL 1,ACC 100,APO_DIST 5,APO_FAC 50.0,ORI_TYP #VAR,CIRC_TYP #BASE,JERK_FAC 50.0}
DECL FDAT FP277={TOOL_NO 2,BASE_NO 10,IPO_FRAME #BASE,POINT2[] " ",TQ_STATE FALSE}
DECL E6POS XP277={X -66.480,Y 122.440,Z -46.660,A 0.000,B -8.000,C -14.990}
DECL LDAT LCPDATC278={VEL 0.1,ACC 100,APO_DIST 5,APO_FAC 50.0,ORI_TYP #VAR,CIRC_TYP #BASE,JERK_FAC 50.0}
DECL FDAT FC278={TOOL_NO 2,BASE_NO 10,IPO_FRAME #BASE,POINT2[] " ",TQ_STATE FALSE}
DECL E6POS XCAux278={X -53.320,Y 128.720,Z -46.660,A -0.000,B -6.410,C -15.720}
DECL E6POS XCDes278={X 53.320,Y 128.720,Z -46.660,A 0.000,B 6.410,C -15.720}
DECL LDAT LCPDATP279={VEL 1,ACC 100,APO_DIST 5,APO_FAC 50.0,ORI_TYP #VAR,CIRC_TYP #BASE,JERK_FAC 50.0}
DECL FDAT FP279={TOOL_NO 2,BASE_NO 10,IPO_FRAME #BASE,POINT2[] " ",TQ_STATE FALSE}
DECL E6POS XP279={X 66.480,Y 122.440,Z -46.660,A -0.000,B 8.000,C -14.990}
DECL LDAT LCPDATP280={VEL 1,ACC 100,APO_DIST 5,APO_FAC 50.0,ORI_TYP #VAR,CIRC_TYP #BASE,JERK_FAC 50.0}
DECL FDAT FP280={TOOL_NO 2,BASE_NO 10,IPO_FRAME #BASE,POINT2[] " ",TQ_STATE FALSE}
DECL E6POS XP280={X 70.240,Y 129.370,Z -48.220,A 0.000,B 2.580,C -4.770}
DECL LDAT LCPDATC281={VEL 0.1,ACC 100,APO_DIST 5,APO_FAC 50.0,ORI_TYP #VAR,CIRC_TYP #BASE,JERK_FAC 50.0}
DECL FDAT FC281={TOOL_NO 2,BASE_NO 10,IPO_FRAME #BASE,POINT2[] " ",TQ_STATE FALSE}
DECL E6POS XCAux281={X 56.340,Y 136.010,Z -48.220,A 0.000,B 2.070,C -5.010}
DECL E6POS XCDes281={X -56.340,Y 136.010,Z -48.220,A -0.000,B -2.070,C -5.010}
DECL LDAT LCPDATP282={VEL 1,ACC 100,APO_DIST 5,APO_FAC 50.0,ORI_TYP #VAR,CIRC_TYP #BASE,JERK_FAC 50.0}
DECL FDAT FP282={TOOL_NO 2,BASE_NO 10,IPO_FRAME #BASE,POINT2[] " ",TQ_STATE FALSE}
DECL E6POS XP282={X -70.240,Y 129.370,Z -48.220,A -0.000,B -2.580,C -4.770}
DECL LDAT LCPDATP283={VEL 1,ACC 100,APO_DIST 5,APO_FAC 50.0,ORI_TYP #VAR,CIRC_TYP #BASE,JERK_FAC 50.0}
DECL FDAT FP283={TOOL_NO 2,BASE_NO 10,IPO_FRAME #BASE,POINT2[] " ",TQ_STATE FALSE}
DECL E6POS XP283={X -71.540,Y 131.770,Z -48.400,A 0.000,B 0.000,C -0.000}
DECL LDAT LCPDATC284={VEL 0.1,ACC 100,APO_DIST 5,APO_FAC 50.0,ORI_TYP #VAR,CIRC_TYP #BASE,JERK_FAC 50.0}
DECL FDAT FC284={TOOL_NO 2,BASE_NO 10,IPO_FRAME #BASE,POINT2[] " ",TQ_STATE FALSE}
DECL E6POS XCAux284={X -57.380,Y 138.530,Z -48.400,A 0.000,B 0.000,C -0.000}
DECL E6POS XCDes284={X 57.380,Y 138.530,Z -48.400,A 0.000,B 0.000,C -0.000}
DECL LDAT LCPDATP285={VEL 1,ACC 100,APO_DIST 5,APO_FAC 50.0,ORI_TYP #VAR,CIRC_TYP #BASE,JERK_FAC 50.0}
DECL FDAT FP285={TOOL_NO 2,BASE_NO 10,IPO_FRAME #BASE,POINT2[] " ",TQ_STATE FALSE}
DECL E6POS XP285={X 71.540,Y 131.770,Z -48.400,A 0.000,B 0.000,C -0.000}
DECL LDAT LCPDATP286={VEL 1,ACC 100,APO_DIST 5,APO_FAC 50.0,ORI_TYP #VAR,CIRC_TYP #BASE,JERK_FAC 50.0}
DECL FDAT FP286={TOOL_NO 2,BASE_NO 10,IPO_FRAME #BASE,POINT2[] " ",TQ_STATE FALSE}
DECL E6POS XP286={X 70.590,Y 130.010,Z -48.400,A 0.000,B 0.000,C -0.000}
DECL LDAT LCPDATC287={VEL 0.1,ACC 100,APO_DIST 5,APO_FAC 50.0,ORI_TYP #VAR,CIRC_TYP #BASE,JERK_FAC 50.0}
DECL FDAT FC287={TOOL_NO 2,BASE_NO 10,IPO_FRAME #BASE,POINT2[] " ",TQ_STATE FALSE}
DECL E6POS XCAux287={X 56.610,Y 136.680,Z -48.400,A 0.000,B 0.000,C -0.000}
DECL E6POS XCDes287={X -56.610,Y 136.680,Z -48.400,A 0.000,B 0.000,C -0.000}
DECL LDAT LCPDATP288={VEL 1,ACC 100,APO_DIST 5,APO_FAC 50.0,ORI_TYP #VAR,CIRC_TYP #BASE,JERK_FAC 50.0}
DECL FDAT FP288={TOOL_NO 2,BASE_NO 10,IPO_FRAME #BASE,POINT2[] " ",TQ_STATE FALSE}
DECL E6POS XP288={X -70.590,Y 130.010,Z -48.400,A 0.000,B 0.000,C -0.000}
DECL LDAT LCPDATP289={VEL 1,ACC 100,APO_DIST 5,APO_FAC 50.0,ORI_TYP #VAR,CIRC_TYP #BASE,JERK_FAC 50.0}
DECL FDAT FP289={TOOL_NO 2,BASE_NO 10,IPO_FRAME #BASE,POINT2[] " ",TQ_STATE FALSE}
DECL E6POS XP289={X -69.640,Y 128.250,Z -48.400,A 0.000,B 0.000,C -0.000}
DECL LDAT LCPDATC290={VEL 0.1,ACC 100,APO_DIST 5,APO_FAC 50.0,ORI_TYP #VAR,CIRC_TYP #BASE,JERK_FAC 50.0}
DECL FDAT FC290={TOOL_NO 2,BASE_NO 10,IPO_FRAME #BASE,POINT2[] " ",TQ_STATE FALSE}
DECL E6POS XCAux290={X -55.850,Y 134.830,Z -48.400,A 0.000,B 0.000,C -0.000}
DECL E6POS XCDes290={X 55.850,Y 134.830,Z -48.400,A 0.000,B 0.000,C -0.000}
DECL LDAT LCPDATP291={VEL 1,ACC 100,APO_DIST 5,APO_FAC 50.0,ORI_TYP #VAR,CIRC_TYP #BASE,JERK_FAC 50.0}
DECL FDAT FP291={TOOL_NO 2,BASE_NO 10,IPO_FRAME #BASE,POINT2[] " ",TQ_STATE FALSE}
DECL E6POS XP291={X 69.640,Y 128.250,Z -48.400,A 0.000,B 0.000,C -0.000}
DECL LDAT LCPDATP292={VEL 1,ACC 100,APO_DIST 5,APO_FAC 50.0,ORI_TYP #VAR,CIRC_TYP #BASE,JERK_FAC 50.0}
DECL FDAT FP292={TOOL_NO 2,BASE_NO 10,IPO_FRAME #BASE,POINT2[] " ",TQ_STATE FALSE}
DECL E6POS XP292={X 68.680,Y 126.500,Z -48.400,A 0.000,B 0.000,C -0.000}
DECL LDAT LCPDATC293={VEL 0.1,ACC 100,APO_DIST 5,APO_FAC 50.0,ORI_TYP #VAR,CIRC_TYP #BASE,JERK_FAC 50.0}
DECL FDAT FC293={TOOL_NO 2,BASE_NO 10,IPO_FRAME #BASE,POINT2[] " ",TQ_STATE FALSE}
DECL E6POS XCAux293={X 55.080,Y 132.980,Z -48.400,A 0.000,B 0.000,C -0.000}
DECL E6POS XCDes293={X -55.080,Y 132.980,Z -48.400,A 0.000,B 0.000,C -0.000}
DECL LDAT LCPDATP294={VEL 1,ACC 100,APO_DIST 5,APO_FAC 50.0,ORI_TYP #VAR,CIRC_TYP #BASE,JERK_FAC 50.0}
DECL FDAT FP294={TOOL_NO 2,BASE_NO 10,IPO_FRAME #BASE,POINT2[] " ",TQ_STATE FALSE}
DECL E6POS XP294={X -68.680,Y 126.500,Z -48.400,A 0.000,B 0.000,C -0.000}
DECL LDAT LCPDATP295={VEL 1,ACC 100,APO_DIST 5,APO_FAC 50.0,ORI_TYP #VAR,CIRC_TYP #BASE,JERK_FAC 50.0}
DECL FDAT FP295={TOOL_NO 2,BASE_NO 10,IPO_FRAME #BASE,POINT2[] " ",TQ_STATE FALSE}
DECL E6POS XP295={X -67.730,Y 124.740,Z -48.400,A 0.000,B 0.000,C -0.000}
DECL LDAT LCPDATC296={VEL 0.1,ACC 100,APO_DIST 5,APO_FAC 50.0,ORI_TYP #VAR,CIRC_TYP #BASE,JERK_FAC 50.0}
DECL FDAT FC296={TOOL_NO 2,BASE_NO 10,IPO_FRAME #BASE,POINT2[] " ",TQ_STATE FALSE}
DECL E6POS XCAux296={X -54.320,Y 131.140,Z -48.400,A 0.000,B 0.000,C -0.000}
DECL E6POS XCDes296={X 54.320,Y 131.140,Z -48.400,A 0.000,B 0.000,C -0.000}
DECL LDAT LCPDATP297={VEL 1,ACC 100,APO_DIST 5,APO_FAC 50.0,ORI_TYP #VAR,CIRC_TYP #BASE,JERK_FAC 50.0}
DECL FDAT FP297={TOOL_NO 2,BASE_NO 10,IPO_FRAME #BASE,POINT2[] " ",TQ_STATE FALSE}
DECL E6POS XP297={X 67.730,Y 124.740,Z -48.400,A 0.000,B 0.000,C -0.000}
DECL LDAT LCPDATP298={VEL 1,ACC 100,APO_DIST 5,APO_FAC 50.0,ORI_TYP #VAR,CIRC_TYP #BASE,JERK_FAC 50.0}
DECL FDAT FP298={TOOL_NO 2,BASE_NO 10,IPO_FRAME #BASE,POINT2[] " ",TQ_STATE FALSE}
DECL E6POS XP298={X 66.770,Y 122.980,Z -48.400,A 0.000,B 0.000,C -0.000}
DECL LDAT LCPDATC299={VEL 0.1,ACC 100,APO_DIST 5,APO_FAC 50.0,ORI_TYP #VAR,CIRC_TYP #BASE,JERK_FAC 50.0}
DECL FDAT FC299={TOOL_NO 2,BASE_NO 10,IPO_FRAME #BASE,POINT2[] " ",TQ_STATE FALSE}
DECL E6POS XCAux299={X 53.550,Y 129.290,Z -48.400,A 0.000,B 0.000,C -0.000}
DECL E6POS XCDes299={X -53.550,Y 129.290,Z -48.400,A 0.000,B 0.000,C -0.000}
DECL LDAT LCPDATP300={VEL 1,ACC 100,APO_DIST 5,APO_FAC 50.0,ORI_TYP #VAR,CIRC_TYP #BASE,JERK_FAC 50.0}
DECL FDAT FP300={TOOL_NO 2,BASE_NO 10,IPO_FRAME #BASE,POINT2[] " ",TQ_STATE FALSE}
DECL E6POS XP300={X -66.770,Y 122.980,Z -48.400,A 0.000,B 0.000,C -0.000}
DECL LDAT LCPDATP301={VEL 1,ACC 100,APO_DIST 5,APO_FAC 50.0,ORI_TYP #VAR,CIRC_TYP #BASE,JERK_FAC 50.0}
DECL FDAT FP301={TOOL_NO 2,BASE_NO 10,IPO_FRAME #BASE,POINT2[] " ",TQ_STATE FALSE}
DECL E6POS XP301={X -68.360,Y 125.910,Z -48.170,A 0.000,B 2.920,C 5.390}
DECL LDAT LCPDATC302={VEL 0.1,ACC 100,APO_DIST 5,APO_FAC 50.0,ORI_TYP #VAR,CIRC_TYP #BASE,JERK_FAC 50.0}
DECL FDAT FC302={TOOL_NO 2,BASE_NO 10,IPO_FRAME #BASE,POINT2[] " ",TQ_STATE FALSE}
DECL E6POS XCAux302={X -54.830,Y 132.370,Z -48.170,A -0.000,B 2.340,C 5.660}
DECL E6POS XCDes302={X 54.830,Y 132.370,Z -48.170,A 0.000,B -2.340,C 5.660}
DECL LDAT LCPDATP303={VEL 1,ACC 100,APO_DIST 5,APO_FAC 50.0,ORI_TYP #VAR,CIRC_TYP #BASE,JERK_FAC 50.0}
DECL FDAT FP303={TOOL_NO 2,BASE_NO 10,IPO_FRAME #BASE,POINT2[] " ",TQ_STATE FALSE}
DECL E6POS XP303={X 68.360,Y 125.910,Z -48.170,A 0.000,B -2.920,C 5.390}
DECL LDAT LCPDATP304={VEL 1,ACC 100,APO_DIST 5,APO_FAC 50.0,ORI_TYP #VAR,CIRC_TYP #BASE,JERK_FAC 50.0}
DECL FDAT FP304={TOOL_NO 2,BASE_NO 10,IPO_FRAME #BASE,POINT2[] " ",TQ_STATE FALSE}
DECL E6POS XP304={X 72.120,Y 132.830,Z -46.510,A 0.000,B -8.320,C 15.620}
DECL LDAT LCPDATC305={VEL 0.1,ACC 100,APO_DIST 5,APO_FAC 50.0,ORI_TYP #VAR,CIRC_TYP #BASE,JERK_FAC 50.0}
DECL FDAT FC305={TOOL_NO 2,BASE_NO 10,IPO_FRAME #BASE,POINT2[] " ",TQ_STATE FALSE}
DECL E6POS XCAux305={X 57.840,Y 139.640,Z -46.510,A 0.000,B -6.660,C 16.380}
DECL E6POS XCDes305={X -57.840,Y 139.640,Z -46.510,A -0.000,B 6.660,C 16.380}
DECL LDAT LCPDATP306={VEL 1,ACC 100,APO_DIST 5,APO_FAC 50.0,ORI_TYP #VAR,CIRC_TYP #BASE,JERK_FAC 50.0}
DECL FDAT FP306={TOOL_NO 2,BASE_NO 10,IPO_FRAME #BASE,POINT2[] " ",TQ_STATE FALSE}
DECL E6POS XP306={X -72.120,Y 132.830,Z -46.510,A 0.000,B 8.320,C 15.620}
DECL LDAT LCPDATP307={VEL 1,ACC 100,APO_DIST 5,APO_FAC 50.0,ORI_TYP #VAR,CIRC_TYP #BASE,JERK_FAC 50.0}
DECL FDAT FP307={TOOL_NO 2,BASE_NO 10,IPO_FRAME #BASE,POINT2[] " ",TQ_STATE FALSE}
DECL E6POS XP307={X -75.640,Y 139.320,Z -43.320,A 0.000,B 13.450,C 26.130}
DECL LDAT LCPDATC308={VEL 0.1,ACC 100,APO_DIST 5,APO_FAC 50.0,ORI_TYP #VAR,CIRC_TYP #BASE,JERK_FAC 50.0}
DECL FDAT FC308={TOOL_NO 2,BASE_NO 10,IPO_FRAME #BASE,POINT2[] " ",TQ_STATE FALSE}
DECL E6POS XCAux308={X -60.670,Y 146.460,Z -43.320,A 0.000,B 10.750,C 27.280}
DECL E6POS XCDes308={X 60.670,Y 146.460,Z -43.320,A 0.000,B -10.750,C 27.280}
DECL LDAT LCPDATP309={VEL 1,ACC 100,APO_DIST 5,APO_FAC 50.0,ORI_TYP #VAR,CIRC_TYP #BASE,JERK_FAC 50.0}
DECL FDAT FP309={TOOL_NO 2,BASE_NO 10,IPO_FRAME #BASE,POINT2[] " ",TQ_STATE FALSE}
DECL E6POS XP309={X 75.640,Y 139.320,Z -43.320,A 0.000,B -13.450,C 26.130}
DECL LDAT LCPDATP310={VEL 1,ACC 100,APO_DIST 5,APO_FAC 50.0,ORI_TYP #VAR,CIRC_TYP #BASE,JERK_FAC 50.0}
DECL FDAT FP310={TOOL_NO 2,BASE_NO 10,IPO_FRAME #BASE,POINT2[] " ",TQ_STATE FALSE}
DECL E6POS XP310={X 78.790,Y 145.110,Z -38.710,A 0.000,B -18.130,C 37.090}
DECL LDAT LCPDATC311={VEL 0.1,ACC 100,APO_DIST 5,APO_FAC 50.0,ORI_TYP #VAR,CIRC_TYP #BASE,JERK_FAC 50.0}
DECL FDAT FC311={TOOL_NO 2,BASE_NO 10,IPO_FRAME #BASE,POINT2[] " ",TQ_STATE FALSE}
DECL E6POS XCAux311={X 63.190,Y 152.550,Z -38.710,A 0.000,B -14.450,C 38.470}
DECL E6POS XCDes311={X -63.190,Y 152.550,Z -38.710,A 0.000,B 14.450,C 38.470}
DECL LDAT LCPDATP312={VEL 1,ACC 100,APO_DIST 5,APO_FAC 50.0,ORI_TYP #VAR,CIRC_TYP #BASE,JERK_FAC 50.0}
DECL FDAT FP312={TOOL_NO 2,BASE_NO 10,IPO_FRAME #BASE,POINT2[] " ",TQ_STATE FALSE}
DECL E6POS XP312={X -78.790,Y 145.110,Z -38.710,A 0.000,B 18.130,C 37.090}
DECL LDAT LCPDATP313={VEL 1,ACC 100,APO_DIST 5,APO_FAC 50.0,ORI_TYP #VAR,CIRC_TYP #BASE,JERK_FAC 50.0}
DECL FDAT FP313={TOOL_NO 2,BASE_NO 10,IPO_FRAME #BASE,POINT2[] " ",TQ_STATE FALSE}
DECL E6POS XP313={X -78.730,Y 145.010,Z -39.330,A -0.000,B 17.860,C 36.410}
DECL LDAT LCPDATC314={VEL 0.1,ACC 100,APO_DIST 5,APO_FAC 50.0,ORI_TYP #VAR,CIRC_TYP #BASE,JERK_FAC 50.0}
DECL FDAT FC314={TOOL_NO 2,BASE_NO 10,IPO_FRAME #BASE,POINT2[] " ",TQ_STATE FALSE}
DECL E6POS XCAux314={X -63.140,Y 152.450,Z -39.330,A -0.000,B 14.240,C 37.780}
DECL E6POS XCDes314={X 63.140,Y 152.450,Z -39.330,A 0.000,B -14.240,C 37.780}
DECL LDAT LCPDATP315={VEL 1,ACC 100,APO_DIST 5,APO_FAC 50.0,ORI_TYP #VAR,CIRC_TYP #BASE,JERK_FAC 50.0}
DECL FDAT FP315={TOOL_NO 2,BASE_NO 10,IPO_FRAME #BASE,POINT2[] " ",TQ_STATE FALSE}
DECL E6POS XP315={X 78.730,Y 145.010,Z -39.330,A -0.000,B -17.860,C 36.410}
DECL LDAT LCPDATP316={VEL 1,ACC 100,APO_DIST 5,APO_FAC 50.0,ORI_TYP #VAR,CIRC_TYP #BASE,JERK_FAC 50.0}
DECL FDAT FP316={TOOL_NO 2,BASE_NO 10,IPO_FRAME #BASE,POINT2[] " ",TQ_STATE FALSE}
DECL E6POS XP316={X 75.390,Y 138.840,Z -44.070,A -0.000,B -12.940,C 25.040}
DECL LDAT LCPDATC317={VEL 0.1,ACC 100,APO_DIST 5,APO_FAC 50.0,ORI_TYP #VAR,CIRC_TYP #BASE,JERK_FAC 50.0}
DECL FDAT FC317={TOOL_NO 2,BASE_NO 10,IPO_FRAME #BASE,POINT2[] " ",TQ_STATE FALSE}
DECL E6POS XCAux317={X 60.460,Y 145.960,Z -44.070,A 0.000,B -10.350,C 26.150}
DECL E6POS XCDes317={X -60.460,Y 145.960,Z -44.070,A 0.000,B 10.350,C 26.150}
DECL LDAT LCPDATP318={VEL 1,ACC 100,APO_DIST 5,APO_FAC 50.0,ORI_TYP #VAR,CIRC_TYP #BASE,JERK_FAC 50.0}
DECL FDAT FP318={TOOL_NO 2,BASE_NO 10,IPO_FRAME #BASE,POINT2[] " ",TQ_STATE FALSE}
DECL E6POS XP318={X -75.390,Y 138.840,Z -44.070,A 0.000,B 12.940,C 25.040}
DECL LDAT LCPDATP319={VEL 1,ACC 100,APO_DIST 5,APO_FAC 50.0,ORI_TYP #VAR,CIRC_TYP #BASE,JERK_FAC 50.0}
DECL FDAT FP319={TOOL_NO 2,BASE_NO 10,IPO_FRAME #BASE,POINT2[] " ",TQ_STATE FALSE}
DECL E6POS XP319={X -71.640,Y 131.950,Z -47.240,A 0.000,B 7.550,C 14.130}
DECL LDAT LCPDATC320={VEL 0.1,ACC 100,APO_DIST 5,APO_FAC 50.0,ORI_TYP #VAR,CIRC_TYP #BASE,JERK_FAC 50.0}
DECL FDAT FC320={TOOL_NO 2,BASE_NO 10,IPO_FRAME #BASE,POINT2[] " ",TQ_STATE FALSE}
DECL E6POS XCAux320={X -57.460,Y 138.710,Z -47.240,A -0.000,B 6.050,C 14.820}
DECL E6POS XCDes320={X 57.460,Y 138.710,Z -47.240,A 0.000,B -6.050,C 14.820}
DECL LDAT LCPDATP321={VEL 1,ACC 100,APO_DIST 5,APO_FAC 50.0,ORI_TYP #VAR,CIRC_TYP #BASE,JERK_FAC 50.0}
DECL FDAT FP321={TOOL_NO 2,BASE_NO 10,IPO_FRAME #BASE,POINT2[] " ",TQ_STATE FALSE}
DECL E6POS XP321={X 71.640,Y 131.950,Z -47.240,A 0.000,B -7.550,C 14.130}
DECL LDAT LCPDATP322={VEL 1,ACC 100,APO_DIST 5,APO_FAC 50.0,ORI_TYP #VAR,CIRC_TYP #BASE,JERK_FAC 50.0}
DECL FDAT FP322={TOOL_NO 2,BASE_NO 10,IPO_FRAME #BASE,POINT2[] " ",TQ_STATE FALSE}
DECL E6POS XP322={X 67.660,Y 124.620,Z -48.700,A 0.000,B -1.890,C 3.490}
DECL LDAT LCPDATC323={VEL 0.1,ACC 100,APO_DIST 5,APO_FAC 50.0,ORI_TYP #VAR,CIRC_TYP #BASE,JERK_FAC 50.0}
DECL FDAT FC323={TOOL_NO 2,BASE_NO 10,IPO_FRAME #BASE,POINT2[] " ",TQ_STATE FALSE}
DECL E6POS XCAux323={X 54.270,Y 131.010,Z -48.700,A 0.000,B -1.520,C 3.670}
DECL E6POS XCDes323={X -54.270,Y 131.010,Z -48.700,A 0.000,B 1.520,C 3.670}
DECL LDAT LCPDATP324={VEL 1,ACC 100,APO_DIST 5,APO_FAC 50.0,ORI_TYP #VAR,CIRC_TYP #BASE,JERK_FAC 50.0}
DECL FDAT FP324={TOOL_NO 2,BASE_NO 10,IPO_FRAME #BASE,POINT2[] " ",TQ_STATE FALSE}
DECL E6POS XP324={X -67.660,Y 124.620,Z -48.700,A 0.000,B 1.890,C 3.490}
